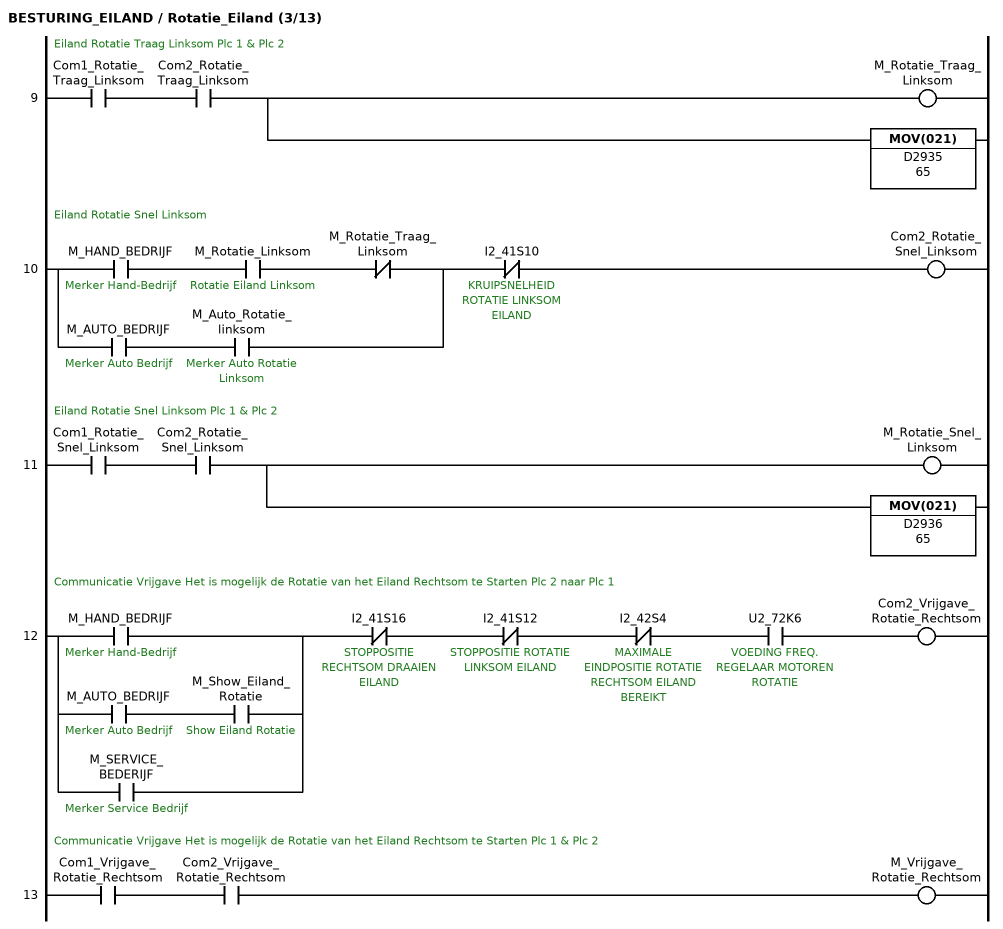
; [picture p421: BESTURING_EILAND / Rotatie_Eiland, rungs 9-13]
; rung 9: Eiland Rotatie Traag Linksom Plc 1 & Plc 2
LD Com1_Rotatie_Traag_Linksom
AND Com2_Rotatie_Traag_Linksom
OUT M_Rotatie_Traag_Linksom
MOV(021) D2935 65
; rung 10: Eiland Rotatie Snel Linksom
LD M_HAND_BEDRIJF  ; Merker Hand-Bedrijf
AND M_Rotatie_Linksom  ; Rotatie Eiland Linksom
ANDNOT M_Rotatie_Traag_Linksom
LD M_AUTO_BEDRIJF  ; Merker Auto Bedrijf
AND M_Auto_Rotatie_linksom  ; Merker Auto Rotatie Linksom
ORLD
ANDNOT I2_41S10  ; KRUIPSNELHEID ROTATIE LINKSOM EILAND
OUT Com2_Rotatie_Snel_Linksom
; rung 11: Eiland Rotatie Snel Linksom Plc 1 & Plc 2
LD Com1_Rotatie_Snel_Linksom
AND Com2_Rotatie_Snel_Linksom
OUT M_Rotatie_Snel_Linksom
MOV(021) D2936 65
; rung 12: Communicatie Vrijgave Het is mogelijk de Rotatie van het Eiland Rechtsom te Starten Plc 2 naar Plc 1
LD M_HAND_BEDRIJF  ; Merker Hand-Bedrijf
LD M_AUTO_BEDRIJF  ; Merker Auto Bedrijf
AND M_Show_Eiland_Rotatie  ; Show Eiland Rotatie
ORLD
OR M_SERVICE_BEDERIJF  ; Merker Service Bedrijf
ANDNOT I2_41S16  ; STOPPOSITIE RECHTSOM DRAAIEN EILAND
ANDNOT I2_41S12  ; STOPPOSITIE ROTATIE LINKSOM EILAND
ANDNOT I2_42S4  ; MAXIMALE EINDPOSITIE ROTATIE RECHTSOM EILAND BEREIKT
AND U2_72K6  ; VOEDING FREQ.REGELAAR MOTOREN ROTATIE
OUT Com2_Vrijgave_Rotatie_Rechtsom
; rung 13: Communicatie Vrijgave Het is mogelijk de Rotatie van het Eiland Rechtsom te Starten Plc 1 & Plc 2
LD Com1_Vrijgave_Rotatie_Rechtsom
AND Com2_Vrijgave_Rotatie_Rechtsom
OUT M_Vrijgave_Rotatie_Rechtsom

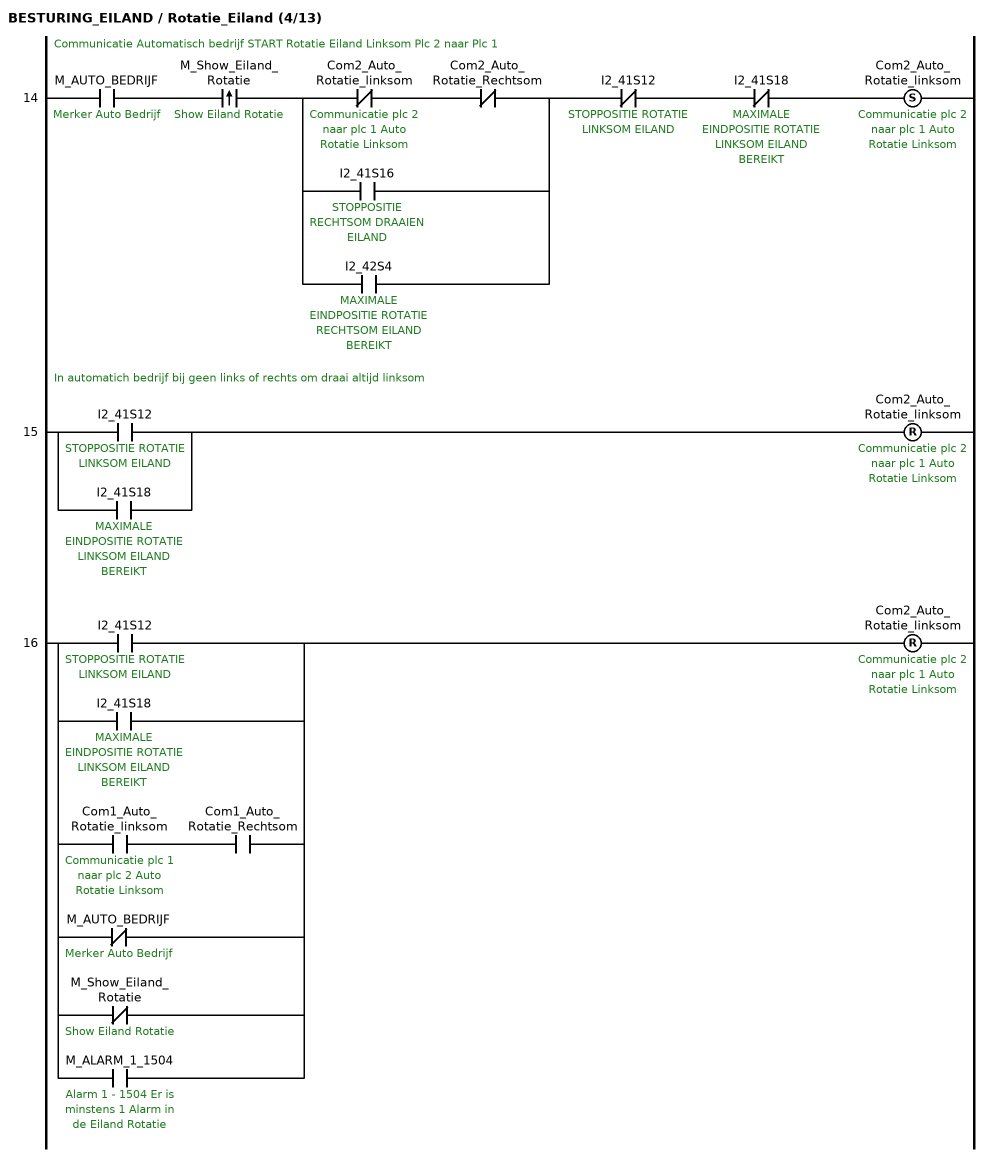
; rung 14: Communicatie Automatisch bedrijf START Rotatie Eiland Linksom Plc 2 naar Plc 1
LD M_AUTO_BEDRIJF  ; Merker Auto Bedrijf
@AND M_Show_Eiland_Rotatie  ; Show Eiland Rotatie
LDNOT Com2_Auto_Rotatie_linksom  ; Communicatie plc 2 naar plc 1 Auto Rotatie Linksom
ANDNOT Com2_Auto_Rotatie_Rechtsom
OR I2_41S16  ; STOPPOSITIE RECHTSOM DRAAIEN EILAND
OR I2_42S4  ; MAXIMALE EINDPOSITIE ROTATIE RECHTSOM EILAND BEREIKT
ANDLD
ANDNOT I2_41S12  ; STOPPOSITIE ROTATIE LINKSOM EILAND
ANDNOT I2_41S18  ; MAXIMALE EINDPOSITIE ROTATIE LINKSOM EILAND BEREIKT
SET Com2_Auto_Rotatie_linksom  ; Communicatie plc 2 naar plc 1 Auto Rotatie Linksom
; rung 15: In automatich bedrijf bij geen links of rechts om draai altijd linksom
LD I2_41S12  ; STOPPOSITIE ROTATIE LINKSOM EILAND
OR I2_41S18  ; MAXIMALE EINDPOSITIE ROTATIE LINKSOM EILAND BEREIKT
RSET Com2_Auto_Rotatie_linksom  ; Communicatie plc 2 naar plc 1 Auto Rotatie Linksom
; rung 16
LD I2_41S12  ; STOPPOSITIE ROTATIE LINKSOM EILAND
OR I2_41S18  ; MAXIMALE EINDPOSITIE ROTATIE LINKSOM EILAND BEREIKT
LD Com1_Auto_Rotatie_linksom  ; Communicatie plc 1 naar plc 2 Auto Rotatie Linksom
AND Com1_Auto_Rotatie_Rechtsom
ORLD
ORNOT M_AUTO_BEDRIJF  ; Merker Auto Bedrijf
ORNOT M_Show_Eiland_Rotatie  ; Show Eiland Rotatie
OR M_ALARM_1_1504  ; Alarm 1 - 1504 Er is minstens 1 Alarm in de Eiland Rotatie
RSET Com2_Auto_Rotatie_linksom  ; Communicatie plc 2 naar plc 1 Auto Rotatie Linksom

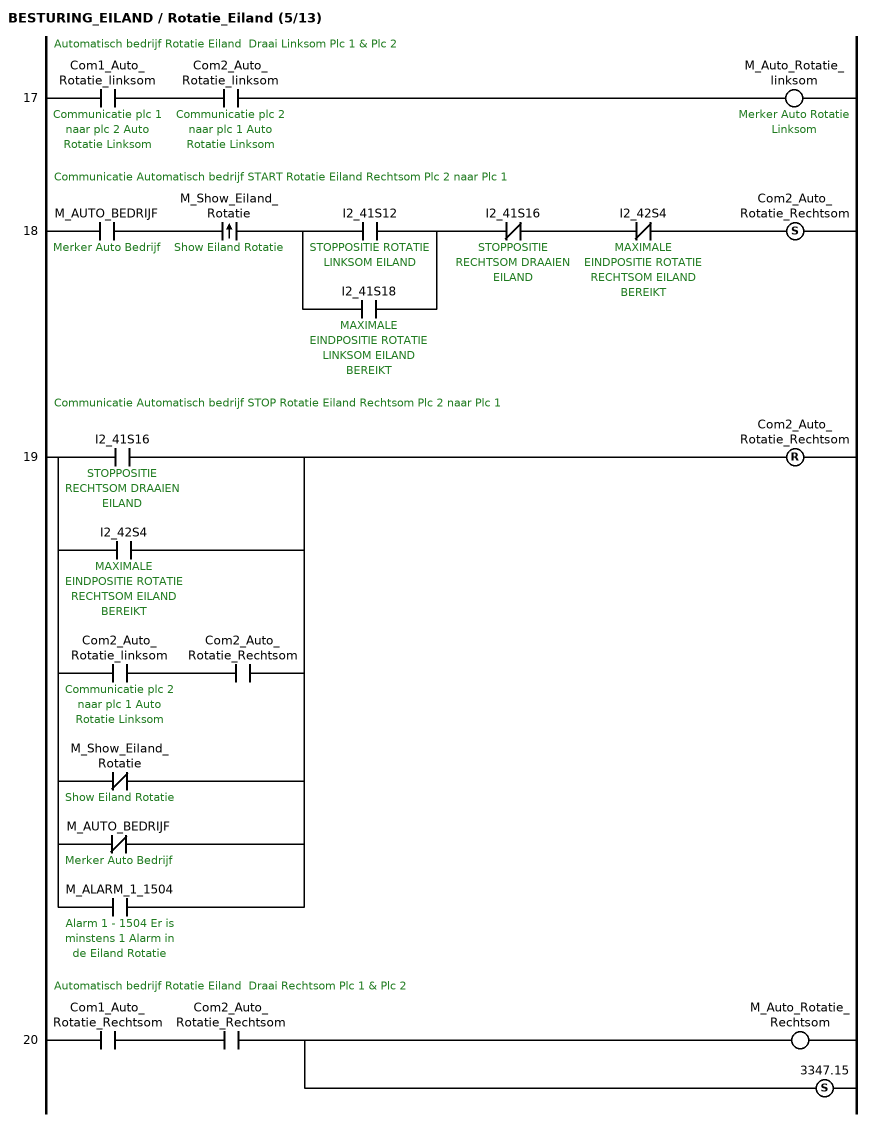
; rung 17: Automatisch bedrijf Rotatie Eiland  Draai Linksom Plc 1 & Plc 2
LD Com1_Auto_Rotatie_linksom  ; Communicatie plc 1 naar plc 2 Auto Rotatie Linksom
AND Com2_Auto_Rotatie_linksom  ; Communicatie plc 2 naar plc 1 Auto Rotatie Linksom
OUT M_Auto_Rotatie_linksom  ; Merker Auto Rotatie Linksom
; rung 18: Communicatie Automatisch bedrijf START Rotatie Eiland Rechtsom Plc 2 naar Plc 1
LD M_AUTO_BEDRIJF  ; Merker Auto Bedrijf
@AND M_Show_Eiland_Rotatie  ; Show Eiland Rotatie
LD I2_41S12  ; STOPPOSITIE ROTATIE LINKSOM EILAND
OR I2_41S18  ; MAXIMALE EINDPOSITIE ROTATIE LINKSOM EILAND BEREIKT
ANDLD
ANDNOT I2_41S16  ; STOPPOSITIE RECHTSOM DRAAIEN EILAND
ANDNOT I2_42S4  ; MAXIMALE EINDPOSITIE ROTATIE RECHTSOM EILAND BEREIKT
SET Com2_Auto_Rotatie_Rechtsom
; rung 19: Communicatie Automatisch bedrijf STOP Rotatie Eiland Rechtsom Plc 2 naar Plc 1
LD I2_41S16  ; STOPPOSITIE RECHTSOM DRAAIEN EILAND
OR I2_42S4  ; MAXIMALE EINDPOSITIE ROTATIE RECHTSOM EILAND BEREIKT
LD Com2_Auto_Rotatie_linksom  ; Communicatie plc 2 naar plc 1 Auto Rotatie Linksom
AND Com2_Auto_Rotatie_Rechtsom
ORLD
ORNOT M_Show_Eiland_Rotatie  ; Show Eiland Rotatie
ORNOT M_AUTO_BEDRIJF  ; Merker Auto Bedrijf
OR M_ALARM_1_1504  ; Alarm 1 - 1504 Er is minstens 1 Alarm in de Eiland Rotatie
RSET Com2_Auto_Rotatie_Rechtsom
; rung 20: Automatisch bedrijf Rotatie Eiland  Draai Rechtsom Plc 1 & Plc 2
LD Com1_Auto_Rotatie_Rechtsom
AND Com2_Auto_Rotatie_Rechtsom
OUT M_Auto_Rotatie_Rechtsom
SET 3347.15

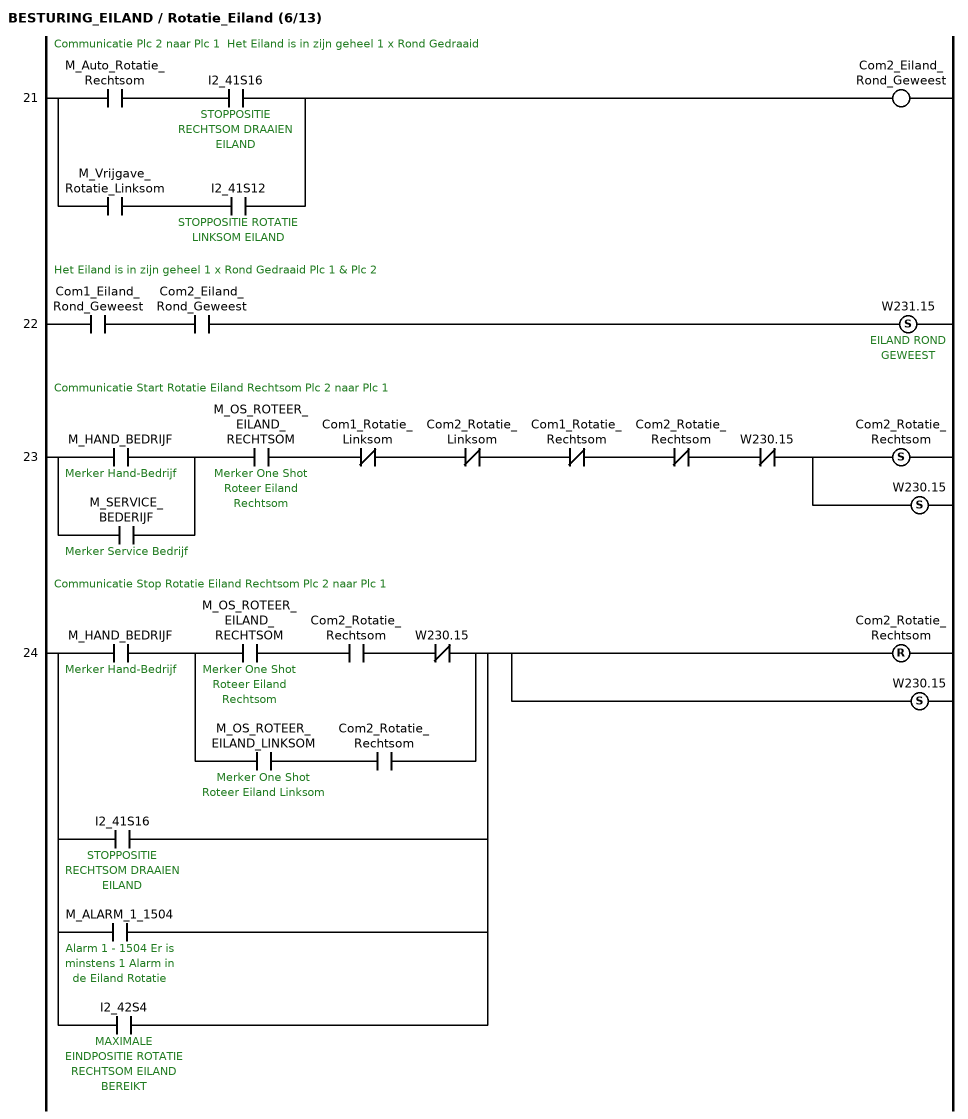
; rung 21: Communicatie Plc 2 naar Plc 1  Het Eiland is in zijn geheel 1 x Rond Gedraaid
LD M_Auto_Rotatie_Rechtsom
AND I2_41S16  ; STOPPOSITIE RECHTSOM DRAAIEN EILAND
LD M_Vrijgave_Rotatie_Linksom
AND I2_41S12  ; STOPPOSITIE ROTATIE LINKSOM EILAND
ORLD
OUT Com2_Eiland_Rond_Geweest
; rung 22: Het Eiland is in zijn geheel 1 x Rond Gedraaid Plc 1 & Plc 2
LD Com1_Eiland_Rond_Geweest
AND Com2_Eiland_Rond_Geweest
SET W231.15  ; EILAND ROND GEWEEST
; rung 23: Communicatie Start Rotatie Eiland Rechtsom Plc 2 naar Plc 1
LD M_HAND_BEDRIJF  ; Merker Hand-Bedrijf
OR M_SERVICE_BEDERIJF  ; Merker Service Bedrijf
AND M_OS_ROTEER_EILAND_RECHTSOM  ; Merker One Shot Roteer Eiland Rechtsom
ANDNOT Com1_Rotatie_Linksom
ANDNOT Com2_Rotatie_Linksom
ANDNOT Com1_Rotatie_Rechtsom
ANDNOT Com2_Rotatie_Rechtsom
ANDNOT W230.15
SET Com2_Rotatie_Rechtsom
SET W230.15
; rung 24: Communicatie Stop Rotatie Eiland Rechtsom Plc 2 naar Plc 1
LD M_HAND_BEDRIJF  ; Merker Hand-Bedrijf
LD M_OS_ROTEER_EILAND_RECHTSOM  ; Merker One Shot Roteer Eiland Rechtsom
AND Com2_Rotatie_Rechtsom
ANDNOT W230.15
LD M_OS_ROTEER_EILAND_LINKSOM  ; Merker One Shot Roteer Eiland Linksom
AND Com2_Rotatie_Rechtsom
ORLD
ANDLD
OR I2_41S16  ; STOPPOSITIE RECHTSOM DRAAIEN EILAND
OR M_ALARM_1_1504  ; Alarm 1 - 1504 Er is minstens 1 Alarm in de Eiland Rotatie
OR I2_42S4  ; MAXIMALE EINDPOSITIE ROTATIE RECHTSOM EILAND BEREIKT
RSET Com2_Rotatie_Rechtsom
SET W230.15

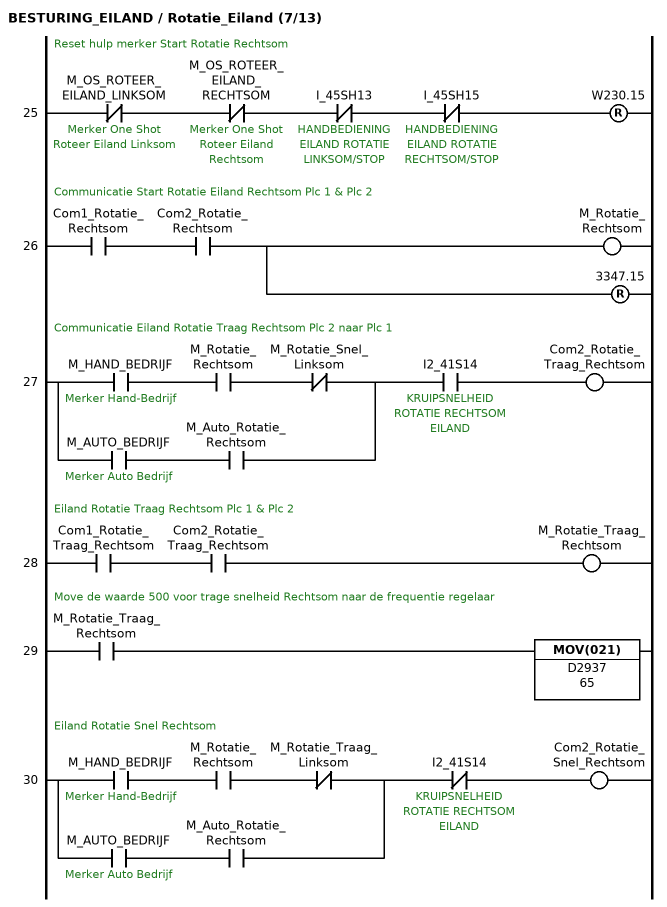
; rung 25: Reset hulp merker Start Rotatie Rechtsom
LDNOT M_OS_ROTEER_EILAND_LINKSOM  ; Merker One Shot Roteer Eiland Linksom
ANDNOT M_OS_ROTEER_EILAND_RECHTSOM  ; Merker One Shot Roteer Eiland Rechtsom
ANDNOT I_45SH13  ; HANDBEDIENING EILAND ROTATIE LINKSOM/STOP
ANDNOT I_45SH15  ; HANDBEDIENING EILAND ROTATIE RECHTSOM/STOP
RSET W230.15
; rung 26: Communicatie Start Rotatie Eiland Rechtsom Plc 1 & Plc 2
LD Com1_Rotatie_Rechtsom
AND Com2_Rotatie_Rechtsom
OUT M_Rotatie_Rechtsom
RSET 3347.15
; rung 27: Communicatie Eiland Rotatie Traag Rechtsom Plc 2 naar Plc 1
LD M_HAND_BEDRIJF  ; Merker Hand-Bedrijf
AND M_Rotatie_Rechtsom
ANDNOT M_Rotatie_Snel_Linksom
LD M_AUTO_BEDRIJF  ; Merker Auto Bedrijf
AND M_Auto_Rotatie_Rechtsom
ORLD
AND I2_41S14  ; KRUIPSNELHEID ROTATIE RECHTSOM EILAND
OUT Com2_Rotatie_Traag_Rechtsom
; rung 28: Eiland Rotatie Traag Rechtsom Plc 1 & Plc 2
LD Com1_Rotatie_Traag_Rechtsom
AND Com2_Rotatie_Traag_Rechtsom
OUT M_Rotatie_Traag_Rechtsom
; rung 29: Move de waarde 500 voor trage snelheid Rechtsom naar de frequentie regelaar
LD M_Rotatie_Traag_Rechtsom
MOV(021) D2937 65
; rung 30: Eiland Rotatie Snel Rechtsom
LD M_HAND_BEDRIJF  ; Merker Hand-Bedrijf
AND M_Rotatie_Rechtsom
ANDNOT M_Rotatie_Traag_Linksom
LD M_AUTO_BEDRIJF  ; Merker Auto Bedrijf
AND M_Auto_Rotatie_Rechtsom
ORLD
ANDNOT I2_41S14  ; KRUIPSNELHEID ROTATIE RECHTSOM EILAND
OUT Com2_Rotatie_Snel_Rechtsom

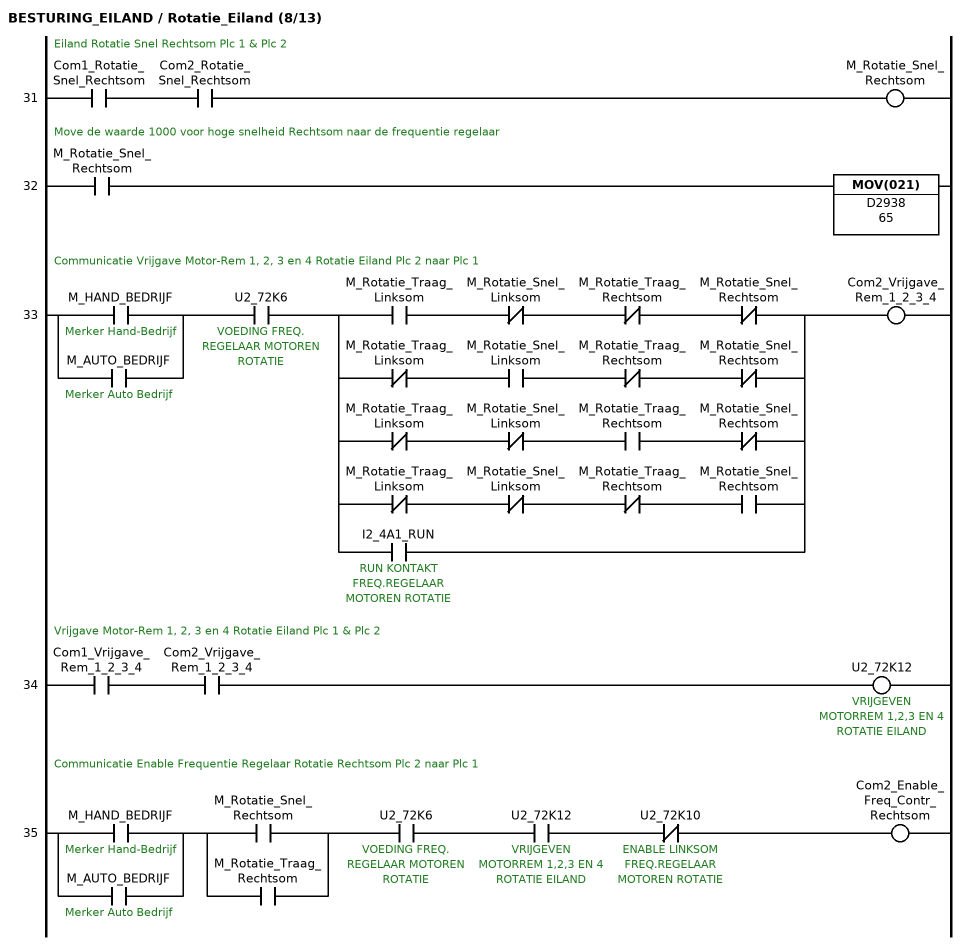
; rung 31: Eiland Rotatie Snel Rechtsom Plc 1 & Plc 2
LD Com1_Rotatie_Snel_Rechtsom
AND Com2_Rotatie_Snel_Rechtsom
OUT M_Rotatie_Snel_Rechtsom
; rung 32: Move de waarde 1000 voor hoge snelheid Rechtsom naar de frequentie regelaar
LD M_Rotatie_Snel_Rechtsom
MOV(021) D2938 65
; rung 33: Communicatie Vrijgave Motor-Rem 1, 2, 3 en 4 Rotatie Eiland Plc 2 naar Plc 1
LD M_HAND_BEDRIJF  ; Merker Hand-Bedrijf
OR M_AUTO_BEDRIJF  ; Merker Auto Bedrijf
AND U2_72K6  ; VOEDING FREQ.REGELAAR MOTOREN ROTATIE
LD M_Rotatie_Traag_Linksom
ANDNOT M_Rotatie_Snel_Linksom
ANDNOT M_Rotatie_Traag_Rechtsom
ANDNOT M_Rotatie_Snel_Rechtsom
LDNOT M_Rotatie_Traag_Linksom
AND M_Rotatie_Snel_Linksom
ANDNOT M_Rotatie_Traag_Rechtsom
ANDNOT M_Rotatie_Snel_Rechtsom
ORLD
LDNOT M_Rotatie_Traag_Linksom
ANDNOT M_Rotatie_Snel_Linksom
AND M_Rotatie_Traag_Rechtsom
ANDNOT M_Rotatie_Snel_Rechtsom
ORLD
LDNOT M_Rotatie_Traag_Linksom
ANDNOT M_Rotatie_Snel_Linksom
ANDNOT M_Rotatie_Traag_Rechtsom
AND M_Rotatie_Snel_Rechtsom
ORLD
OR I2_4A1_RUN  ; RUN KONTAKT FREQ.REGELAAR MOTOREN ROTATIE
ANDLD
OUT Com2_Vrijgave_Rem_1_2_3_4
; rung 34: Vrijgave Motor-Rem 1, 2, 3 en 4 Rotatie Eiland Plc 1 & Plc 2
LD Com1_Vrijgave_Rem_1_2_3_4
AND Com2_Vrijgave_Rem_1_2_3_4
OUT U2_72K12  ; VRIJGEVEN MOTORREM 1,2,3 EN 4 ROTATIE EILAND
; rung 35: Communicatie Enable Frequentie Regelaar Rotatie Rechtsom Plc 2 naar Plc 1
LD M_HAND_BEDRIJF  ; Merker Hand-Bedrijf
OR M_AUTO_BEDRIJF  ; Merker Auto Bedrijf
LD M_Rotatie_Snel_Rechtsom
OR M_Rotatie_Traag_Rechtsom
ANDLD
AND U2_72K6  ; VOEDING FREQ.REGELAAR MOTOREN ROTATIE
AND U2_72K12  ; VRIJGEVEN MOTORREM 1,2,3 EN 4 ROTATIE EILAND
ANDNOT U2_72K10  ; ENABLE LINKSOM FREQ.REGELAAR MOTOREN ROTATIE
OUT Com2_Enable_Freq_Contr_Rechtsom

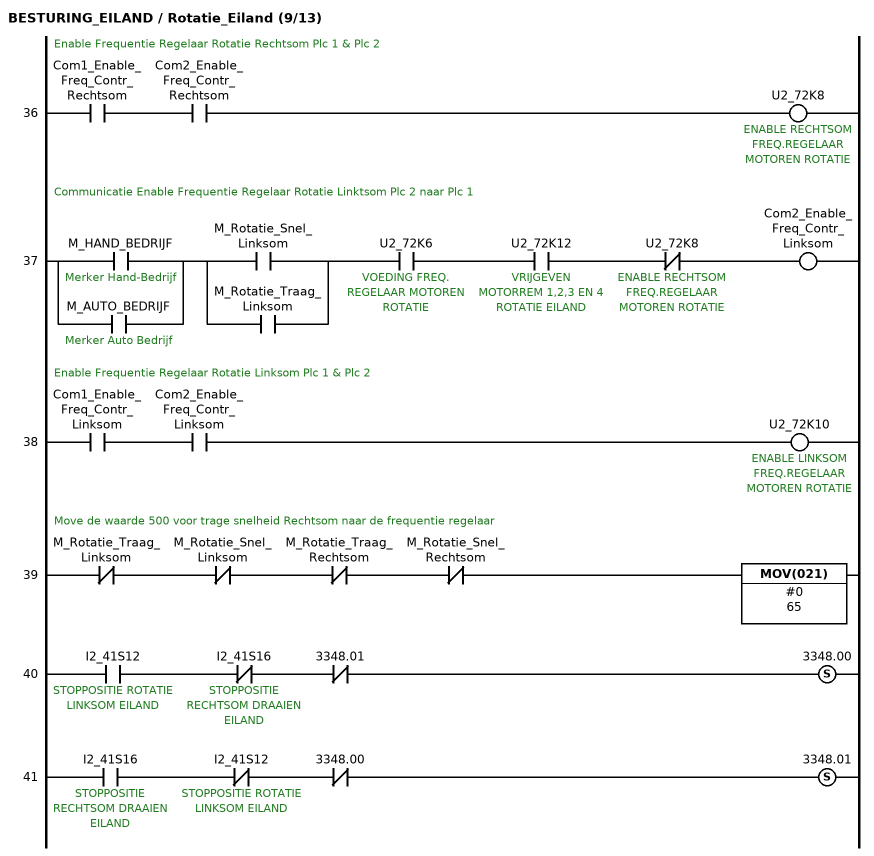
; rung 36: Enable Frequentie Regelaar Rotatie Rechtsom Plc 1 & Plc 2
LD Com1_Enable_Freq_Contr_Rechtsom
AND Com2_Enable_Freq_Contr_Rechtsom
OUT U2_72K8  ; ENABLE RECHTSOM FREQ.REGELAAR MOTOREN ROTATIE
; rung 37: Communicatie Enable Frequentie Regelaar Rotatie Linktsom Plc 2 naar Plc 1
LD M_HAND_BEDRIJF  ; Merker Hand-Bedrijf
OR M_AUTO_BEDRIJF  ; Merker Auto Bedrijf
LD M_Rotatie_Snel_Linksom
OR M_Rotatie_Traag_Linksom
ANDLD
AND U2_72K6  ; VOEDING FREQ.REGELAAR MOTOREN ROTATIE
AND U2_72K12  ; VRIJGEVEN MOTORREM 1,2,3 EN 4 ROTATIE EILAND
ANDNOT U2_72K8  ; ENABLE RECHTSOM FREQ.REGELAAR MOTOREN ROTATIE
OUT Com2_Enable_Freq_Contr_Linksom
; rung 38: Enable Frequentie Regelaar Rotatie Linksom Plc 1 & Plc 2
LD Com1_Enable_Freq_Contr_Linksom
AND Com2_Enable_Freq_Contr_Linksom
OUT U2_72K10  ; ENABLE LINKSOM FREQ.REGELAAR MOTOREN ROTATIE
; rung 39: Move de waarde 500 voor trage snelheid Rechtsom naar de frequentie regelaar
LDNOT M_Rotatie_Traag_Linksom
ANDNOT M_Rotatie_Snel_Linksom
ANDNOT M_Rotatie_Traag_Rechtsom
ANDNOT M_Rotatie_Snel_Rechtsom
MOV(021) #0 65
; rung 40
LD I2_41S12  ; STOPPOSITIE ROTATIE LINKSOM EILAND
ANDNOT I2_41S16  ; STOPPOSITIE RECHTSOM DRAAIEN EILAND
ANDNOT 3348.01
SET 3348.00
; rung 41
LD I2_41S16  ; STOPPOSITIE RECHTSOM DRAAIEN EILAND
ANDNOT I2_41S12  ; STOPPOSITIE ROTATIE LINKSOM EILAND
ANDNOT 3348.00
SET 3348.01

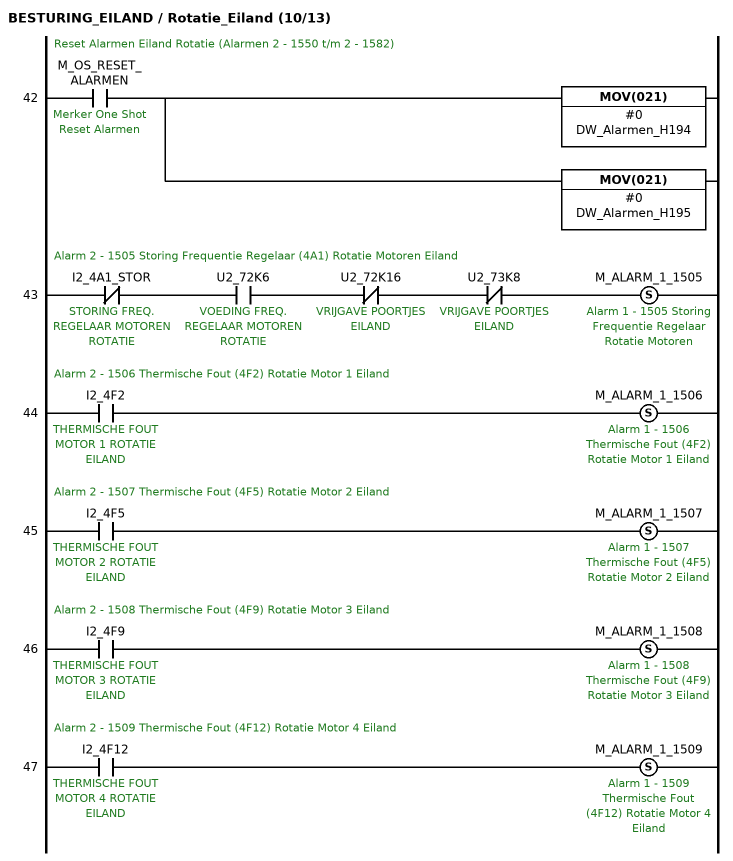
; rung 42: Reset Alarmen Eiland Rotatie (Alarmen 2 - 1550 t/m 2 - 1582)
LD M_OS_RESET_ALARMEN  ; Merker One Shot Reset Alarmen
MOV(021) #0 DW_Alarmen_H194
MOV(021) #0 DW_Alarmen_H195
; rung 43: Alarm 2 - 1505 Storing Frequentie Regelaar (4A1) Rotatie Motoren Eiland
LDNOT I2_4A1_STOR  ; STORING FREQ.REGELAAR MOTOREN ROTATIE
AND U2_72K6  ; VOEDING FREQ.REGELAAR MOTOREN ROTATIE
ANDNOT U2_72K16  ; VRIJGAVE POORTJES EILAND
ANDNOT U2_73K8  ; VRIJGAVE POORTJES EILAND
SET M_ALARM_1_1505  ; Alarm 1 - 1505 Storing Frequentie Regelaar Rotatie Motoren
; rung 44: Alarm 2 - 1506 Thermische Fout (4F2) Rotatie Motor 1 Eiland
LD I2_4F2  ; THERMISCHE FOUT MOTOR 1 ROTATIE EILAND
SET M_ALARM_1_1506  ; Alarm 1 - 1506 Thermische Fout (4F2) Rotatie Motor 1 Eiland
; rung 45: Alarm 2 - 1507 Thermische Fout (4F5) Rotatie Motor 2 Eiland
LD I2_4F5  ; THERMISCHE FOUT MOTOR 2 ROTATIE EILAND
SET M_ALARM_1_1507  ; Alarm 1 - 1507 Thermische Fout (4F5) Rotatie Motor 2 Eiland
; rung 46: Alarm 2 - 1508 Thermische Fout (4F9) Rotatie Motor 3 Eiland
LD I2_4F9  ; THERMISCHE FOUT MOTOR 3 ROTATIE EILAND
SET M_ALARM_1_1508  ; Alarm 1 - 1508 Thermische Fout (4F9) Rotatie Motor 3 Eiland
; rung 47: Alarm 2 - 1509 Thermische Fout (4F12) Rotatie Motor 4 Eiland
LD I2_4F12  ; THERMISCHE FOUT MOTOR 4 ROTATIE EILAND
SET M_ALARM_1_1509  ; Alarm 1 - 1509 Thermische Fout (4F12) Rotatie Motor 4 Eiland

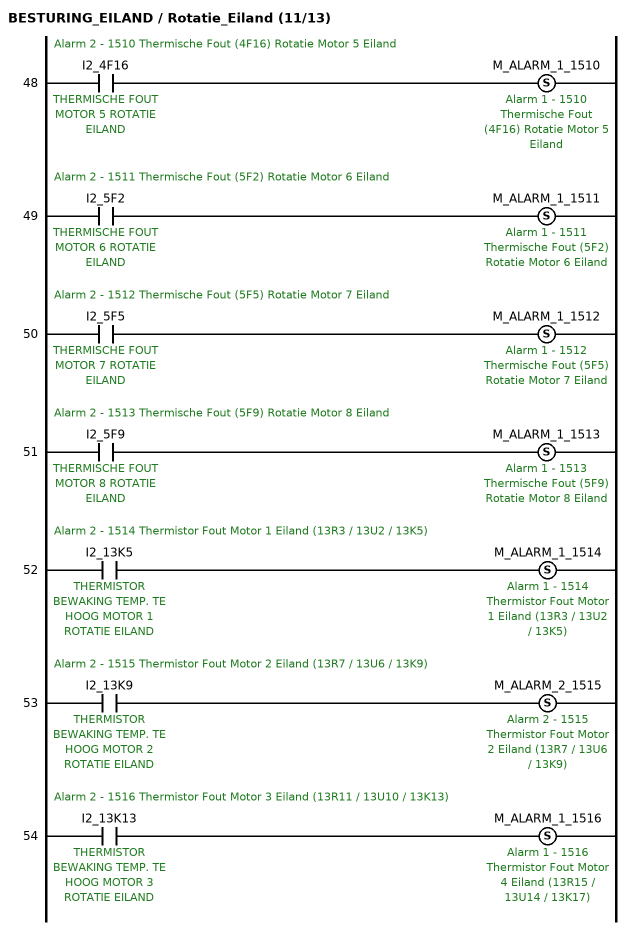
; rung 48: Alarm 2 - 1510 Thermische Fout (4F16) Rotatie Motor 5 Eiland
LD I2_4F16  ; THERMISCHE FOUT MOTOR 5 ROTATIE EILAND
SET M_ALARM_1_1510  ; Alarm 1 - 1510 Thermische Fout (4F16) Rotatie Motor 5 Eiland
; rung 49: Alarm 2 - 1511 Thermische Fout (5F2) Rotatie Motor 6 Eiland
LD I2_5F2  ; THERMISCHE FOUT MOTOR 6 ROTATIE EILAND
SET M_ALARM_1_1511  ; Alarm 1 - 1511 Thermische Fout (5F2) Rotatie Motor 6 Eiland
; rung 50: Alarm 2 - 1512 Thermische Fout (5F5) Rotatie Motor 7 Eiland
LD I2_5F5  ; THERMISCHE FOUT MOTOR 7 ROTATIE EILAND
SET M_ALARM_1_1512  ; Alarm 1 - 1512 Thermische Fout (5F5) Rotatie Motor 7 Eiland
; rung 51: Alarm 2 - 1513 Thermische Fout (5F9) Rotatie Motor 8 Eiland
LD I2_5F9  ; THERMISCHE FOUT MOTOR 8 ROTATIE EILAND
SET M_ALARM_1_1513  ; Alarm 1 - 1513 Thermische Fout (5F9) Rotatie Motor 8 Eiland
; rung 52: Alarm 2 - 1514 Thermistor Fout Motor 1 Eiland (13R3 / 13U2 / 13K5)
LD I2_13K5  ; THERMISTOR BEWAKING TEMP. TE HOOG MOTOR 1 ROTATIE EILAND
SET M_ALARM_1_1514  ; Alarm 1 - 1514 Thermistor Fout Motor 1 Eiland (13R3 / 13U2 / 13K5)
; rung 53: Alarm 2 - 1515 Thermistor Fout Motor 2 Eiland (13R7 / 13U6 / 13K9)
LD I2_13K9  ; THERMISTOR BEWAKING TEMP. TE HOOG MOTOR 2 ROTATIE EILAND
SET M_ALARM_2_1515  ; Alarm 2 - 1515 Thermistor Fout Motor 2 Eiland (13R7 / 13U6 / 13K9)
; rung 54: Alarm 2 - 1516 Thermistor Fout Motor 3 Eiland (13R11 / 13U10 / 13K13)
LD I2_13K13  ; THERMISTOR BEWAKING TEMP. TE HOOG MOTOR 3 ROTATIE EILAND
SET M_ALARM_1_1516  ; Alarm 1 - 1516 Thermistor Fout Motor 4 Eiland (13R15 / 13U14 / 13K17)

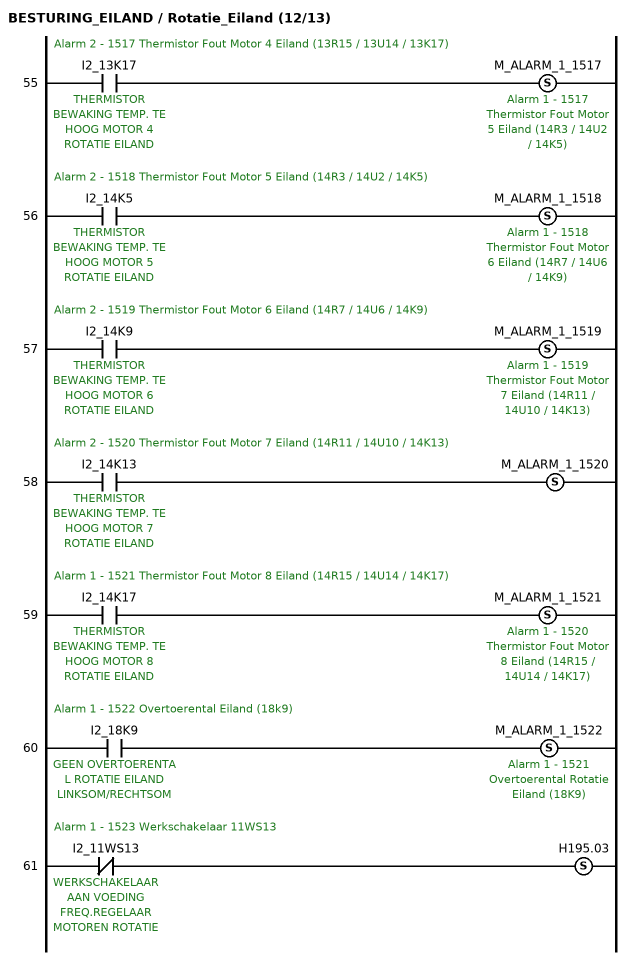
; rung 55: Alarm 2 - 1517 Thermistor Fout Motor 4 Eiland (13R15 / 13U14 / 13K17)
LD I2_13K17  ; THERMISTOR BEWAKING TEMP. TE HOOG MOTOR 4 ROTATIE EILAND
SET M_ALARM_1_1517  ; Alarm 1 - 1517 Thermistor Fout Motor 5 Eiland (14R3 / 14U2 / 14K5)
; rung 56: Alarm 2 - 1518 Thermistor Fout Motor 5 Eiland (14R3 / 14U2 / 14K5)
LD I2_14K5  ; THERMISTOR BEWAKING TEMP. TE HOOG MOTOR 5 ROTATIE EILAND
SET M_ALARM_1_1518  ; Alarm 1 - 1518 Thermistor Fout Motor 6 Eiland (14R7 / 14U6 / 14K9)
; rung 57: Alarm 2 - 1519 Thermistor Fout Motor 6 Eiland (14R7 / 14U6 / 14K9)
LD I2_14K9  ; THERMISTOR BEWAKING TEMP. TE HOOG MOTOR 6 ROTATIE EILAND
SET M_ALARM_1_1519  ; Alarm 1 - 1519 Thermistor Fout Motor 7 Eiland (14R11 / 14U10 / 14K13)
; rung 58: Alarm 2 - 1520 Thermistor Fout Motor 7 Eiland (14R11 / 14U10 / 14K13)
LD I2_14K13  ; THERMISTOR BEWAKING TEMP. TE HOOG MOTOR 7 ROTATIE EILAND
SET M_ALARM_1_1520
; rung 59: Alarm 1 - 1521 Thermistor Fout Motor 8 Eiland (14R15 / 14U14 / 14K17)
LD I2_14K17  ; THERMISTOR BEWAKING TEMP. TE HOOG MOTOR 8 ROTATIE EILAND
SET M_ALARM_1_1521  ; Alarm 1 - 1520 Thermistor Fout Motor 8 Eiland (14R15 / 14U14 / 14K17)
; rung 60: Alarm 1 - 1522 Overtoerental Eiland (18k9)
LD I2_18K9  ; GEEN OVERTOERENTAL ROTATIE EILAND LINKSOM/RECHTSOM
SET M_ALARM_1_1522  ; Alarm 1 - 1521 Overtoerental Rotatie Eiland (18K9)
; rung 61: Alarm 1 - 1523 Werkschakelaar 11WS13
LDNOT I2_11WS13  ; WERKSCHAKELAAR AAN VOEDING FREQ.REGELAAR MOTOREN ROTATIE
SET H195.03

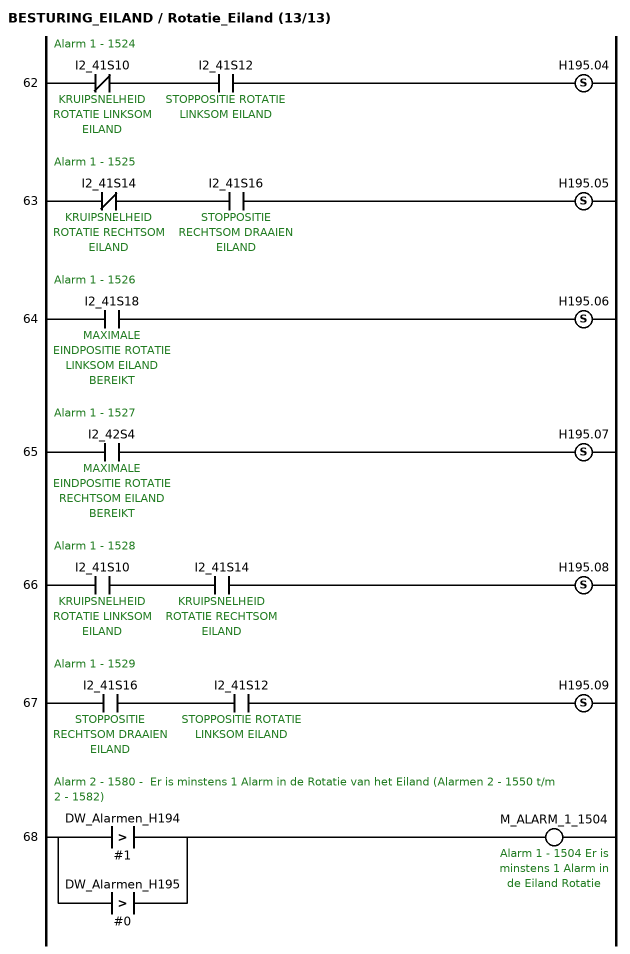
; rung 62: Alarm 1 - 1524
LDNOT I2_41S10  ; KRUIPSNELHEID ROTATIE LINKSOM EILAND
AND I2_41S12  ; STOPPOSITIE ROTATIE LINKSOM EILAND
SET H195.04
; rung 63: Alarm 1 - 1525
LDNOT I2_41S14  ; KRUIPSNELHEID ROTATIE RECHTSOM EILAND
AND I2_41S16  ; STOPPOSITIE RECHTSOM DRAAIEN EILAND
SET H195.05
; rung 64: Alarm 1 - 1526
LD I2_41S18  ; MAXIMALE EINDPOSITIE ROTATIE LINKSOM EILAND BEREIKT
SET H195.06
; rung 65: Alarm 1 - 1527
LD I2_42S4  ; MAXIMALE EINDPOSITIE ROTATIE RECHTSOM EILAND BEREIKT
SET H195.07
; rung 66: Alarm 1 - 1528
LD I2_41S10  ; KRUIPSNELHEID ROTATIE LINKSOM EILAND
AND I2_41S14  ; KRUIPSNELHEID ROTATIE RECHTSOM EILAND
SET H195.08
; rung 67: Alarm 1 - 1529
LD I2_41S16  ; STOPPOSITIE RECHTSOM DRAAIEN EILAND
AND I2_41S12  ; STOPPOSITIE ROTATIE LINKSOM EILAND
SET H195.09
; rung 68: Alarm 2 - 1580 -  Er is minstens 1 Alarm in de Rotatie van het Eiland (Alarmen 2 - 1550 t/m 2 - 1582)
LD>(320) DW_Alarmen_H194 #1
OR>(320) DW_Alarmen_H195 #0
OUT M_ALARM_1_1504  ; Alarm 1 - 1504 Er is minstens 1 Alarm in de Eiland Rotatie

### Section EInde_Besturing_Eiland
; rung 0
END(001)

# PLC PLC3_PAGODE_EILAND: CJ2M CPU12
I/O table (CPU CJ2M-CPU12): rack 0 slot 0 CJ1W-CLK23; rack 0 slot 1 CJ1W-ID211; rack 0 slot 2 CJ1W-ID211; rack 0 slot 3 CJ1W-ID211; rack 0 slot 4 CJ1W-ID211; rack 0 slot 5 CJ1W-OD212; rack 0 slot 6 CJ1W-OD212; rack 0 slot 7 CJ1W-OD212

## Global symbols (name address type ; comment)
ALL_24_VDC_RELAY_ON 230.03 BOOL  ; ALL 24 VDC RELAY ON
102.01 BOOL  ; show afbreken
102.02 BOOL  ; noodberging 1
102.03 BOOL  ; noodberging 2
125.03 BOOL  ; Signalering stop show vanaf grond
217.00 BOOL  ; Alarm in register 0 zoeken
217.01 BOOL  ; Alarm in register 1 zoeken
217.02 BOOL  ; Alarm in register 2 zoeken
217.03 BOOL  ; Alarm in register 3 zoeken
217.04 BOOL  ; Alarm in register 4 zoeken
217.05 BOOL  ; Alarm in register 5 zoeken
217.08 BOOL  ; Alarm (1 of meerdere)
217.09 BOOL  ; Alarmlamp knipperen bij nieuw alarm
217.10 BOOL  ; Zoeken naar nieuw alarm
217.11 BOOL  ; Volgend alarmwoord bekijken
217.12 BOOL  ; Alarm zoeken in volgende woord
217.13 BOOL  ; Volgende alarm gevonden
217.14 BOOL  ; Elke 2 seconden 1 scan hoog
217.15 BOOL  ; Zoek volgende alarm melding
218.08 BOOL  ; Nieuw alarm in woord HR30
218.09 BOOL  ; Nieuw alarm in woord HR31
218.10 BOOL  ; Nieuw alarm in woord HR32
218.11 BOOL  ; Nieuw alarm in woord HR33
218.12 BOOL  ; Nieuw alarm in woord HR34
218.13 BOOL  ; Nieuw alarm in woord HR35
218.14 BOOL  ; Geen nieuw alarm
218.15 BOOL  ; 1 scan, er is een nieuw alarm opgetreden
219.00 BOOL  ; Alarm in register 6 zoeken
219.01 BOOL  ; Alarm in register 7 zoeken
219.02 BOOL  ; Alarm in register 8 zoeken
219.03 BOOL  ; Alarm in register 8 zoeken
219.08 BOOL  ; Nieuw alarm in woord HR36
219.09 BOOL  ; Nieuw alarm in woord HR37
219.10 BOOL  ; Nieuw alarm in woord HR38
219.11 BOOL  ; Alle poorten staan dicht
224.00 BOOL  ; Poort 1 links is open
224.01 BOOL  ; Poort 1 links is dicht
224.02 BOOL  ; Poort 1 links is aan het openen
224.03 BOOL  ; Poort 1 links is aan het sluiten
224.04 BOOL  ; Poort 1 rechts is open
224.05 BOOL  ; Poort 1 rechts is dicht
224.06 BOOL  ; Poort 1 rechts is aan het openen
224.07 BOOL  ; Poort 1 rechts is aan het sluiten
224.08 BOOL  ; Poort 2 links is open
224.09 BOOL  ; Poort 2 links is dicht
224.10 BOOL  ; Poort 2 links is aan het openen
224.11 BOOL  ; poort 2 links is aan het sluiten
224.12 BOOL  ; Poort 2 rechts is open
224.13 BOOL  ; Poort 2 rechts is dicht
224.14 BOOL  ; Poort 2 rechts is aan het openen
224.15 BOOL  ; Poort 2 rechts is aan het sluiten
225.00 BOOL  ; Poort 3 links is open
225.01 BOOL  ; Poort 3 links is dicht
225.02 BOOL  ; Poort 3 links is aan het openen
225.03 BOOL  ; Poort 3 links is aan het sluiten
225.04 BOOL  ; Poort 3 rechts is open
225.05 BOOL  ; Poort 3 rechts is dicht
225.06 BOOL  ; Poort 3 rechts is aan het openen
225.07 BOOL  ; Poort 3 rechts is aan het sluiten
225.08 BOOL  ; Poort 4 links is open
225.09 BOOL  ; Poort 4 links is dicht
225.10 BOOL  ; Poort 4 links is aan het openen
225.11 BOOL  ; Poort 4 links is aan het sluiten
225.12 BOOL  ; Poort 4 rechts is open
225.13 BOOL  ; Poort 4 rechts is dicht
225.14 BOOL  ; Poort 4 rechts is aan het openen
225.15 BOOL  ; Poort 4 rechts is aan het sluiten
230.04 BOOL  ; stop show
232.02 BOOL  ; stop van grond
240.01 BOOL  ; Testmerker
T0100 BOOL  ; DISPATCH TIMER
T0101 BOOL  ; TIMER 24 VDC RELAY 01 (ALL RELAY ON)
T0102 BOOL  ; TIMER 24 VDC RELAY 02 (ONE RELAY OFF)
DISPATCH_ACTIVE 231.00 BOOL  ; DISPATCH ACTIVE
DISPATCH_ISLAND_ENABLE 230.00 BOOL  ; DISPATCH ISLAND ENABLE
DISPATCH_TIMER 100 NUMBER  ; DISPATCH TIMER
DISPATCH_TIMER_ACTIVE 230.02 BOOL  ; DISPATCH TIMER ACTIVE
I1L_BEWAK 2.08 BOOL  ; POORT 1 LINKS BEWAKING
I1L_BIJNA 0.07 BOOL  ; POORT 1 LINKS BIJNA DICHT
I1L_DICHT 0.06 BOOL  ; POORT 1 LINKS DICHT
I1L_GREND 2.00 BOOL  ; POORT 1 LINKS VERGRENDELD
I1L_OPEN 0.08 BOOL  ; POORT 1 LINKS OPEN
I1R_BEWAK 2.09 BOOL  ; POORT 1 RECHTS BEWAKING
I1R_BIJNA 0.10 BOOL  ; POORT 1 RECHTS BIJNA DICHT
I1R_DICHT 0.09 BOOL  ; POORT 1 RECHTS DICHT
I1R_GREND 2.01 BOOL  ; POORT 1 RECHTS VERGRENDELD
I1R_OPEN 0.11 BOOL  ; POORT 1 RECHTS OPEN
I24V_OKE1 3.00 BOOL  ; 24 VOLT OKE (MELDING 1)
I24V_OKE2 3.01 BOOL  ; 24 VOLT OKE (MELDING 2)
I24V_OKE3 3.02 BOOL  ; 24 VOLT OKE (MELDING 3)
I2L_BEWAK 2.10 BOOL  ; POORT 2 LINKS BEWAKING
I2L_BIJNA 0.13 BOOL  ; POORT 2 LINKS BIJNA DICHT
I2L_DICHT 0.12 BOOL  ; POORT 2 LINKS DICHT
I2L_GREND 2.02 BOOL  ; POORT 2 LINKS VERGRENDELD
I2L_OPEN 0.14 BOOL  ; POORT 2 LINKS OPEN
I2R_BEWAK 2.11 BOOL  ; POORT 2 RECHTS BEWAKING
I2R_BIJNA 1.00 BOOL  ; POORT 2 RECHTS BIJNA DICHT
I2R_DICHT 0.15 BOOL  ; POORT 2 RECHTS DICHT
I2R_GREND 2.03 BOOL  ; POORT 2 RECHTS VERGRENDELD
I2R_OPEN 1.01 BOOL  ; POORT 2 RECHTS OPEN
I3L_BEWAK 2.12 BOOL  ; POORT 3 LINKS BEWAKING
I3L_BIJNA 1.03 BOOL  ; POORT 3 LINKS  BIJNA DICHT
I3L_DICHT 1.02 BOOL  ; POORT 3 LINKS  DICHT
I3L_GREND 2.04 BOOL  ; POORT 3 LINKS VERGRENDELD
I3L_OPEN 1.04 BOOL  ; POORT 3 LINKS  OPEN
I3R_BEWAK 2.13 BOOL  ; POORT 3 RECHTS BEWAKING
I3R_BIJNA 1.06 BOOL  ; POORT 3 RECHTS BIJNA DICHT
I3R_DICHT 1.05 BOOL  ; POORT 3 RECHTS DICHT
I3R_GREND 2.05 BOOL  ; POORT 3 RECHTS VERGRENDELD
I3R_OPEN 1.07 BOOL  ; POORT 3 RECHTS OPEN
I4L_BEWAK 2.14 BOOL  ; POORT 4 LINKS BEWAKING
I4L_BIJNA 1.09 BOOL  ; POORT 4 LINKS BIJNA DICHT
I4L_DICHT 1.08 BOOL  ; POORT 4 LINKS DICHT
I4L_GREND 2.06 BOOL  ; POORT 4 LINKS VERGRENDELD
I4L_OPEN 1.10 BOOL  ; POORT 4 LINKS OPEN
I4R_BEWAK 2.15 BOOL  ; POORT 4 RECHTS BEWAKING
I4R_BIJNA 1.12 BOOL  ; POORT 4 RECHTS BIJNA DICHT
I4R_DICHT 1.11 BOOL  ; POORT 4 RECHTS DICHT
I4R_GREND 2.07 BOOL  ; POORT 4 RECHTS VERGRENDELD
I4R_OPEN 1.13 BOOL  ; POORT 4 RECHTS OPEN
IAUTOMAAT 0.05 BOOL  ; AUTOMAAT VOEDINGS GROEP MOTOREN
INIT_BIT A200.15 BOOL  ; FIRST SCAN BIT
INOODSTOP 0.00 BOOL  ; NOODSTOP OKE
IOPEN_IN 0.01 BOOL  ; DK OPENEN POORTEN INGANG
IOPEN_UI 0.03 BOOL  ; DK OPENEN POORTEN UITGANG
IREADY 1.14 BOOL  ; DK READY SIGNAAL
IRESET 1.15 BOOL  ; DK RESET
ISLUIT_IN 0.02 BOOL  ; DK SLUITEN POORTEN INGANG
ISLUIT_UI 0.04 BOOL  ; DK SLUITEN POORTEN UITGANG
M1SECPULS CF102 BOOL  ; 1 SEC. HOOG, 1 SEC LAAG = 0,5 HZ
MAL19909 27.09 BOOL  ; OUTPUT ALARM RESERVE BIT
MAL19910 27.10 BOOL  ; OUTPUT ALARM RESERVE BIT
MAL19911 27.11 BOOL  ; OUTPUT ALARM RESERVE BIT
MAL19912 27.12 BOOL  ; OUTPUT ALARM RESERVE BIT
MAL19913 27.13 BOOL  ; OUTPUT ALARM RESEREV BIT
MAL19914 27.14 BOOL  ; OUTPUT ALARM RESEREV BIT
MAL19915 27.15 BOOL  ; OUTPUT ALARM RESERVE BIT
MALBEWAK 27.08 BOOL  ; ALARM BEWAKING AANGESPROKEN
MALM9909 23.09 BOOL  ; ALARM RESERVE BIT
MALM9910 23.10 BOOL  ; ALARM RESERVE BIT
MALM9911 23.11 BOOL  ; ALARM RESERVE BIT
MALM9912 23.12 BOOL  ; ALARM RESERVE BIT
MALM9913 23.13 BOOL  ; ALARM RESERVE BIT
MALM9914 23.14 BOOL  ; ALARM RESERVE BIT
MALM9915 23.15 BOOL  ; ALARM RESERVE BIT
MALMBIJ1 27.04 BOOL  ; ALARM BIJNA OPEN SENSOR 1
MALMBIJ2 27.05 BOOL  ; ALARM BIJNA OPEN SENSOR 2
MALMDI1 27.06 BOOL  ; ALARM DICHT SENSOR 1
MALMDI2 27.07 BOOL  ; ALARM DICHT SENSOR 2
MALMNOODS H30.00 BOOL  ; ALARM NOODSTOP
MALMOP1 27.02 BOOL  ; ALARM OPEN SENSOR 1
MALMOP2 27.03 BOOL  ; ALARM OPEN SENSOR 2
MALMPAL1 27.00 BOOL  ; PAL ALARM 1
MALMPAL2 27.01 BOOL  ; PAL ALARM 2
MALMW0 170.00 BOOL  ; ALARM IN WOORD HR 30
MALMW1 170.01 BOOL  ; ALARM IN WOORD HR 31
MALMW2 170.02 BOOL  ; ALARM IN WOORD HR 32
MALMW3 170.03 BOOL  ; ALARM IN WOORD HR 33
MALMW4 170.04 BOOL  ; ALARM IN WOORD HR 34
MALMW5 170.05 BOOL  ; ALARM IN WOORD HR 35
MALMW6 170.06 BOOL  ; ALARM IN WOORD HR 36
MALMW7 170.07 BOOL  ; ALARM IN WOORD HR 37
MALMW8 170.08 BOOL  ; ALARM IN WOORD HR 38
MALM_BIJ1 23.04 BOOL  ; ALARM BIJNA OPEN SENSOR 1
MALM_BIJ2 23.05 BOOL  ; ALARM BIJNA OPEN SENSOR 2
MALM_DI1 23.06 BOOL  ; ALARM DICHT SENSOR 1
MALM_DI2 23.07 BOOL  ; ALARM DICHT SENSOR 2
MALM_OP1 23.02 BOOL  ; ALARM OPEN SENSOR 1
MALM_OP2 23.03 BOOL  ; ALARM OPEN SENSOR 2
MALM_PAL1 23.00 BOOL  ; ALARM PAL 1
MALM_PAL2 23.01 BOOL  ; ALARM PAL 2
MALTIJD1 CF113 BOOL  ; SYSTEEMBIT ALTIJD 1
MAL_BEWAK 23.08 BOOL  ; ALARM BEWAKING AANGESPROKEN
MAUTOMAAT H30.01 BOOL  ; ALARM INSTALLATIE AUTOMAAT
MBIT0TMR 26.00 BOOL  ; BIT 0 PRESET STAP TIMER
MBIT10TMR 26.10 BOOL  ; BIT 10 PRESET STAP TIMER
MBIT11TMR 26.11 BOOL  ; BIT 11PRESET STAP TIMER
MBIT12TMR 26.12 BOOL  ; BIT 12 PRESET STAP TIMER
MBIT13TMR 26.13 BOOL  ; BIT 13 PRESET STAP TIMER
MBIT14TMR 26.14 BOOL  ; BIT 14 PRESET STAP TIMER
MBIT15TMR 26.15 BOOL  ; BIT 15 PRESET STAP TIMER
MBIT1TMR 26.01 BOOL  ; BIT 1 PRESET STAP TIMER
MBIT2TMR 26.02 BOOL  ; BIT 2 PRESET STAP TIMER
MBIT3TMR 26.03 BOOL  ; BIT 3 PRESET STAP TIMER
MBIT4TMR 26.04 BOOL  ; BIT 4 PRESET STAP TIMER
MBIT5TMR 26.05 BOOL  ; BIT 5 PRESET STAP TIMER
MBIT6TMR 26.06 BOOL  ; BIT 6 PRESET STAP TIMER
MBIT7TMR 26.07 BOOL  ; BIT 7 PRESET STAP TIMER
MBIT8TMR 26.08 BOOL  ; BIT 8 PRESET STAP TIMER
MBIT9TMR 26.09 BOOL  ; BIT 9 PRESET STAP TIMER
MBLINKER CF101 BOOL  ; BLINK MERKER 5 HZ
MDOORTOEG 25.15 BOOL  ; DOORSTAP TOEGESTAAN
MGELIJK CF006 BOOL  ; IS GELIJK AAN
MI_STAP0 21.00 BOOL  ; STAP 0 (SUB)
MI_STAP1 21.01 BOOL  ; STAP 1 (SUB)
MI_STAP10 21.10 BOOL  ; STAP 10 (SUB)
MI_STAP11 21.11 BOOL  ; STAP 11 (SUB)
MI_STAP12 21.12 BOOL  ; STAP 12 (SUB)
MI_STAP13 21.13 BOOL  ; STAP 13 (SUB)
MI_STAP14 21.14 BOOL  ; STAP 14 (SUB)
MI_STAP15 21.15 BOOL  ; STAP 15 (SUB)
MI_STAP2 21.02 BOOL  ; STAP 2 (SUB)
MI_STAP3 21.03 BOOL  ; STAP 3 (SUB)
MI_STAP4 21.04 BOOL  ; STAP 4 (SUB)
MI_STAP5 21.05 BOOL  ; STAP 5 (SUB)
MI_STAP6 21.06 BOOL  ; STAP 6 (SUB)
MI_STAP7 21.07 BOOL  ; STAP 7 (SUB)
MI_STAP8 21.08 BOOL  ; STAP 8 (SUB)
MI_STAP9 21.09 BOOL  ; STAP 9 (SUB)
MMOTOR_O 24.00 BOOL  ; MOTOR OPENEN (SUB)
MMOTOR_S 24.01 BOOL  ; MOTOR SLUITEN (SUB)
MOSYSTOKE 24.12 BOOL  ; SYSTEEM OKE
MO_STAP0 25.00 BOOL  ; OUTPUT STAP  0 (SUB)
MO_STAP1 25.01 BOOL  ; OUTPUT STAP 1 (SUB)
MO_STAP10 25.10 BOOL  ; OUTPUT STAP 10 (SUB)
MO_STAP11 25.11 BOOL  ; OUTPUT STAP 11 (SUB)
MO_STAP12 25.12 BOOL  ; OUTPUT STAP 12 (SUB)
MO_STAP13 25.13 BOOL  ; OUTPUT STAP 13 (SUB)
MO_STAP14 25.14 BOOL  ; OUTPUT STAP 14 (SUB)
MO_STAP2 25.02 BOOL  ; OUTPUT STAP 2 (SUB)
MO_STAP3 25.03 BOOL  ; OUTPUT STAP 3 (SUB)
MO_STAP4 25.04 BOOL  ; OUTPUT STAP 4 (SUB)
MO_STAP5 25.05 BOOL  ; OUTPUT STAP 5 (SUB)
MO_STAP6 25.06 BOOL  ; OUTPUT STAP 6 (SUB)
MO_STAP7 25.07 BOOL  ; OUTPUT STAP 7  (SUB)
MO_STAP8 25.08 BOOL  ; OUTPUT STAP 8  (SUB)
MO_STAP9 25.09 BOOL  ; OUTPUT STAP 9 (SUB)
MPRTDICHT 24.04 BOOL  ; POORT  IS DICHT
MPRTOPEN 24.03 BOOL  ; POORT  IS OPEN
M_OPENT 24.05 BOOL  ; POORT  IS AAN HET OPENEN
M_PAL 24.02 BOOL  ; PAL OMHOOG STUREN (SUB)
M_SLUIT 24.06 BOOL  ; POORT IS AAN HET SLUITEN
O1L_GREND 101.00 BOOL  ; POORT 1 LINKS VERGRENDELEN
O1L_OPEN 100.00 BOOL  ; POORT 1 LINKS OPENEN
O1L_SLUIT 100.01 BOOL  ; POORT 1 LINKS SLUITEN
O1R_GREND 101.01 BOOL  ; POORT 1 RECHTS VERGRENDELEN
O1R_OPEN 100.02 BOOL  ; POORT 1 RECHTS OPENEN
O1R_SLUIT 100.03 BOOL  ; POORT 1 RECHTS SLUITEN
O2L_GREND 101.02 BOOL  ; POORT 2 LINKS  VERGRENDELEN
O2L_OPEN 100.04 BOOL  ; POORT 2 LINKS OPENEN
O2L_SLUIT 100.05 BOOL  ; POORT 2 LINKS SLUITEN
O2R_GREND 101.03 BOOL  ; POORT 2 RECHTS VERGRENDELEN
O2R_OPEN 100.06 BOOL  ; POORT 2 RECHTS OPENEN
O2R_SLUIT 100.07 BOOL  ; POORT 2 RECHTS SLUITEN
O3L_GREND 101.04 BOOL  ; POORT 3 LINKS VERGRENDELEN
O3L_OPEN 100.08 BOOL  ; POORT 3 LINKS OPENEN
O3L_SLUIT 100.09 BOOL  ; POORT 3 LINKS SLUITEN
O3R_GREND 101.05 BOOL  ; POORT 3 RECHTS VERGRENDELEN
O3R_OPEN 100.10 BOOL  ; POORT 3 RECHTS OPENEN
O3R_SLUIT 100.11 BOOL  ; POORT 3 RECHTS SLUITEN
O4L_GREND 101.06 BOOL  ; POORT 4 LINKS VERGRENDELEN
O4L_OPEN 100.12 BOOL  ; POORT 4 LINKS OPENEN
O4L_SLUIT 100.13 BOOL  ; POORT 4 LINKS SLUITEN
O4R_GREND 101.07 BOOL  ; POORT 4 RECHTS VERGRENDELEN
O4R_OPEN 100.14 BOOL  ; POORT 4 RECHTS OPENEN
O4R_SLUIT 100.15 BOOL  ; POORT 4 RECHTS SLUITEN
O514 101.14 BOOL  ; RESERVE UITGANG 514
O515 101.15 BOOL  ; RESERVE UITGANG 515
OH_IDICHT 101.11 BOOL  ; LAMP POORTJES INGANG DICHT
OH_IOPEN 101.10 BOOL  ; LAMP POORTJES INGANG GEOPEND
OH_READY 101.09 BOOL  ; LAMP READY SIGNAAL
OH_UDICHT 101.13 BOOL  ; LAMP POORTJES UITGANG DICHT
OH_UOPEN 101.12 BOOL  ; LAMP POORTJES UITGANG GEOPEND
OREADY 101.08 BOOL  ; READY SIGNAAL
RALM0OUD D460 CHANNEL  ; REG. ALARM HR 30 VORIGE SCAN
RALM1OUD D461 CHANNEL  ; REG. ALARM HR 31 VORIGE SCAN
RALM2OUD D462 CHANNEL  ; REG. ALARM HR32 VORIGE SCAN
RALM3OUD D463 CHANNEL  ; REG. ALARM HR 33 VORIGE SCAN
RALM4OUD D464 CHANNEL  ; REG. ALARM HR 34 VORIGE SCAN
RALM5OUD D465 CHANNEL  ; REG. ALARM HR 35 VORIGE SCAN
RALM6OUD D466 CHANNEL  ; REG. ALARM HR 36 VORIGE SCAN
RALM7OUD D467 CHANNEL  ; REG. ALARM HR 37 VORIGE SCAN
RALM8OUD D468 CHANNEL  ; REG. ALARM HR 38 VORIGE SCAN
RALMTEMP D459 CHANNEL  ; HULP REG. ALARM
RDALNMR D453 CHANNEL  ; REG. DISPLAY ALARMNUMMER BCD
RDSCHUIF D450 CHANNEL  ; REG. DISPLAY SCHUIFREGISTER
RDTELLER D451 CHANNEL  ; REG. DISPLAY 1 T/M 16
RRALMAKT D452 CHANNEL  ; REG. CONTROLE OF ER IN 1 WOORD EEN ALARM HOOG IS
S9602 96.02 BOOL  ; RESERVE
S9603 96.03 BOOL  ; RESERVE
SOPENEN 20.00 BOOL  ; OPENEN IN/UITGANG (SUB)
SRESET 20.04 BOOL  ; DK RESET BEDIEND (SUB)
SSLUITEN 20.01 BOOL  ; SLUITEN IN/UITGANG (SUB)
SSYSTOKE 20.13 BOOL  ; SYSTEEM OKE (SUB)
START_PULSE 230.01 BOOL  ; START PULSE FROM PUSH BUTTON
S_ALTIJD1 20.14 BOOL  ; ALTIJD 1 BIT  (SUB)
S_BEWAK 20.09 BOOL  ; POORT BEWAKING  (SUB)
S_BIJNA 20.06 BOOL  ; POORT BIJNA DICHT (SUB)
S_DICHT 20.05 BOOL  ; POORT DICHT (SUB)
S_GREND 20.08 BOOL  ; POORT VERGRENDELD  (SUB)
S_OPEN 20.07 BOOL  ; POORT OPEN (SUB)
S_TIMER 20.15 BOOL  ; STAPPENTIMER AFGELOPEN (SUB)
TDISPLAY_PV T206 CHANNEL  ; TIMER OVERBRUG DISPLAY WAARDE
TDISPLAY_Status T0206 BOOL  ; TIMER OVERBRUG DISPLAY WAARDE
TDISPSCRO_PV T207 CHANNEL  ; SCROLLEN ALARMS DISPLAY
TDISPSCRO_Status T0207 BOOL  ; SCROLLEN ALARMS DISPLAY
TIMER_24_VDC_RELAY_01 101 NUMBER  ; TIMER 24 VDC RELAY 01 (ALL RELAY ON)
TIMER_24_VDC_RELAY_02 102 NUMBER  ; TIMER 24 VDC RELAY 02 (ONE RELAY OFF)
TMR_PRG1_PV T31 CHANNEL  ; STAPPENTIMER POORT 1 LINKS
TMR_PRG1_Status T0031 BOOL  ; STAPPENTIMER POORT 1 LINKS
TMR_PRG2_PV T32 CHANNEL  ; STAPPENTIMER POORT 1 RECHTS
TMR_PRG2_Status T0032 BOOL  ; STAPPENTIMER POORT 1 RECHTS
TMR_PRG3_PV T33 CHANNEL  ; STAPPENTIMER POORT 2 LINKS
TMR_PRG3_Status T0033 BOOL  ; STAPPENTIMER POORT 2 LINKS
TMR_PRG4_PV T34 CHANNEL  ; STAPPENTIMER POORT 2 RECHTS
TMR_PRG4_Status T0034 BOOL  ; STAPPENTIMER POORT 2 RECHTS
TMR_PRG5_PV T35 CHANNEL  ; STAPPENTIMER POORT 3 LINKS
TMR_PRG5_Status T0035 BOOL  ; STAPPENTIMER POORT 3 LINKS
TMR_PRG6_PV T36 CHANNEL  ; STAPPENTIMER POORT 3 RECHTS
TMR_PRG6_Status T0036 BOOL  ; STAPPENTIMER POORT 3 RECHTS
TMR_PRG7_PV T37 CHANNEL  ; STAPPENTIMER POORT 4 LINKS
TMR_PRG7_Status T0037 BOOL  ; STAPPENTIMER POORT 4 LINKS
TMR_PRG8_PV T38 CHANNEL  ; STAPPENTIMER POORT 4 RECHTS
TMR_PRG8_Status T0038 BOOL  ; STAPPENTIMER POORT 4 RECHTS
com3_afbreek_show 130.03 BOOL  ; com 3 afbreken show
stop_show 3.03 BOOL  ; afbreken running show

## Program POORTEN (cyclic task 0)
Local symbols
Com3_Alarm_in_Plc3 130.01 BOOL  ; Er is minstens 1 alarm in plc 3 eiland poortjes
Com3_Open_Oever_Poortjes 130.00 BOOL
DK_Open_Oever_Poortjes 3.05 BOOL  ; Open Oever Poortjes

### Section algemeen
; rung 0: PAGODE / *************************************************************************** / Projekt: PAGODE, Besturing poorten        Proj.nr. LvH: 760114 / Locatie: Efteling, Kaatsheuvel. / ***************************************************************************

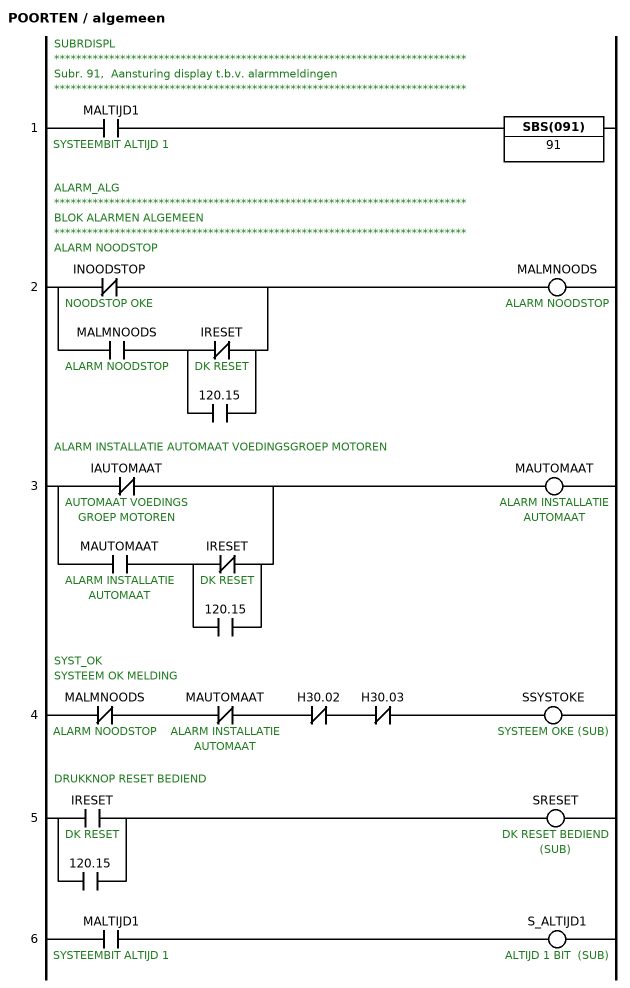
; rung 1: SUBRDISPL / *************************************************************************** / Subr. 91,  Aansturing display t.b.v. alarmmeldingen / ***************************************************************************
LD MALTIJD1  ; SYSTEEMBIT ALTIJD 1
SBS(091) 91
; rung 2: ALARM_ALG / *************************************************************************** / BLOK ALARMEN ALGEMEEN / *************************************************************************** / ALARM NOODSTOP
LDNOT INOODSTOP  ; NOODSTOP OKE
LD MALMNOODS  ; ALARM NOODSTOP
LDNOT IRESET  ; DK RESET
OR 120.15
ANDLD
ORLD
OUT MALMNOODS  ; ALARM NOODSTOP
; rung 3: ALARM INSTALLATIE AUTOMAAT VOEDINGSGROEP MOTOREN
LDNOT IAUTOMAAT  ; AUTOMAAT VOEDINGS GROEP MOTOREN
LD MAUTOMAAT  ; ALARM INSTALLATIE AUTOMAAT
LDNOT IRESET  ; DK RESET
OR 120.15
ANDLD
ORLD
OUT MAUTOMAAT  ; ALARM INSTALLATIE AUTOMAAT
; rung 4: SYST_OK / SYSTEEM OK MELDING
LDNOT MALMNOODS  ; ALARM NOODSTOP
ANDNOT MAUTOMAAT  ; ALARM INSTALLATIE AUTOMAAT
ANDNOT H30.02
ANDNOT H30.03
OUT SSYSTOKE  ; SYSTEEM OKE (SUB)
; rung 5: DRUKKNOP RESET BEDIEND
LD IRESET  ; DK RESET
OR 120.15
OUT SRESET  ; DK RESET BEDIEND (SUB)
; rung 6
LD MALTIJD1  ; SYSTEEMBIT ALTIJD 1
OUT S_ALTIJD1  ; ALTIJD 1 BIT  (SUB)

### Section CONTROL_LINK

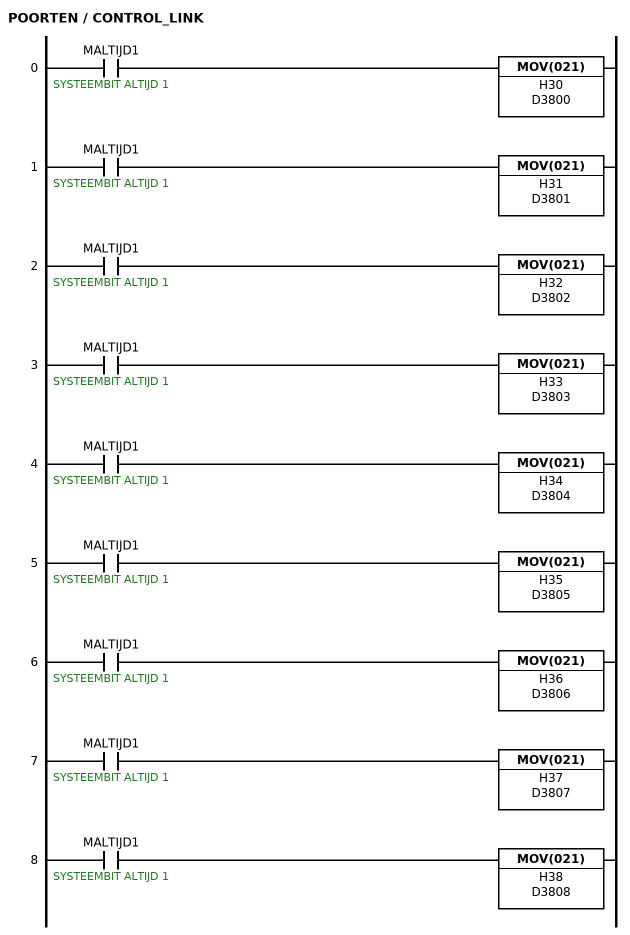
; rung 0
LD MALTIJD1  ; SYSTEEMBIT ALTIJD 1
MOV(021) H30 D3800
; rung 1
LD MALTIJD1  ; SYSTEEMBIT ALTIJD 1
MOV(021) H31 D3801
; rung 2
LD MALTIJD1  ; SYSTEEMBIT ALTIJD 1
MOV(021) H32 D3802
; rung 3
LD MALTIJD1  ; SYSTEEMBIT ALTIJD 1
MOV(021) H33 D3803
; rung 4
LD MALTIJD1  ; SYSTEEMBIT ALTIJD 1
MOV(021) H34 D3804
; rung 5
LD MALTIJD1  ; SYSTEEMBIT ALTIJD 1
MOV(021) H35 D3805
; rung 6
LD MALTIJD1  ; SYSTEEMBIT ALTIJD 1
MOV(021) H36 D3806
; rung 7
LD MALTIJD1  ; SYSTEEMBIT ALTIJD 1
MOV(021) H37 D3807
; rung 8
LD MALTIJD1  ; SYSTEEMBIT ALTIJD 1
MOV(021) H38 D3808

### Section SIGNAAL_DISPLAY

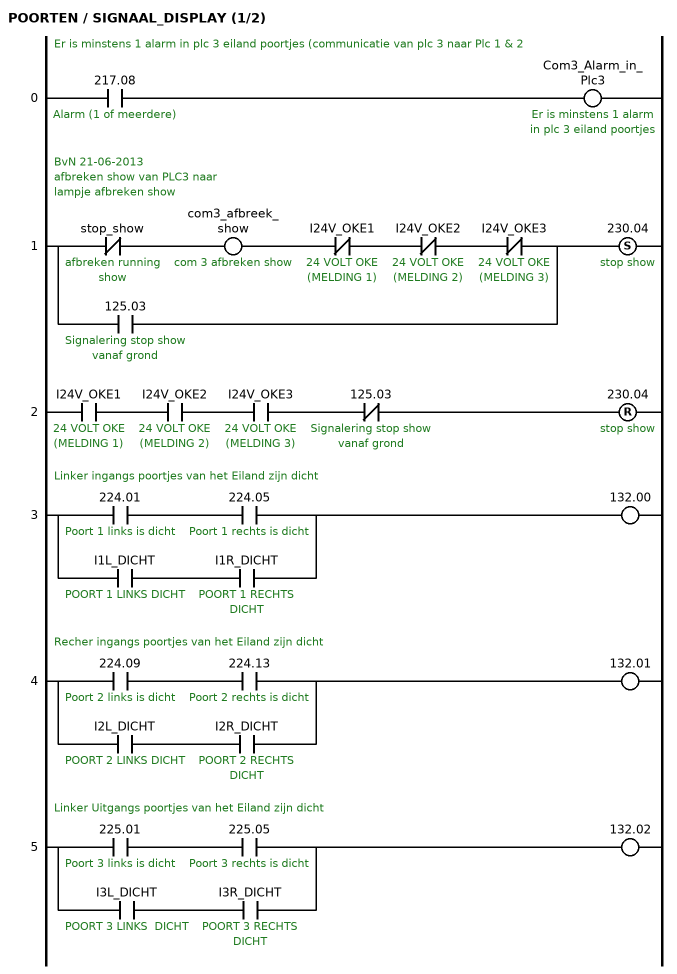
; rung 0: Er is minstens 1 alarm in plc 3 eiland poortjes (communicatie van plc 3 naar Plc 1 & 2
LD 217.08  ; Alarm (1 of meerdere)
OUT Com3_Alarm_in_Plc3  ; Er is minstens 1 alarm in plc 3 eiland poortjes
; rung 1: BvN 21-06-2013 / afbreken show van PLC3 naar / lampje afbreken show
LDNOT stop_show  ; afbreken running show
OUT com3_afbreek_show  ; com 3 afbreken show
ANDNOT I24V_OKE1  ; 24 VOLT OKE (MELDING 1)
ANDNOT I24V_OKE2  ; 24 VOLT OKE (MELDING 2)
ANDNOT I24V_OKE3  ; 24 VOLT OKE (MELDING 3)
OR 125.03  ; Signalering stop show vanaf grond
SET 230.04  ; stop show
; rung 2
LD I24V_OKE1  ; 24 VOLT OKE (MELDING 1)
AND I24V_OKE2  ; 24 VOLT OKE (MELDING 2)
AND I24V_OKE3  ; 24 VOLT OKE (MELDING 3)
ANDNOT 125.03  ; Signalering stop show vanaf grond
RSET 230.04  ; stop show
; rung 3: Linker ingangs poortjes van het Eiland zijn dicht
LD 224.01  ; Poort 1 links is dicht
AND 224.05  ; Poort 1 rechts is dicht
LD I1L_DICHT  ; POORT 1 LINKS DICHT
AND I1R_DICHT  ; POORT 1 RECHTS DICHT
ORLD
OUT 132.00
; rung 4: Recher ingangs poortjes van het Eiland zijn dicht
LD 224.09  ; Poort 2 links is dicht
AND 224.13  ; Poort 2 rechts is dicht
LD I2L_DICHT  ; POORT 2 LINKS DICHT
AND I2R_DICHT  ; POORT 2 RECHTS DICHT
ORLD
OUT 132.01
; rung 5: Linker Uitgangs poortjes van het Eiland zijn dicht
LD 225.01  ; Poort 3 links is dicht
AND 225.05  ; Poort 3 rechts is dicht
LD I3L_DICHT  ; POORT 3 LINKS  DICHT
AND I3R_DICHT  ; POORT 3 RECHTS DICHT
ORLD
OUT 132.02

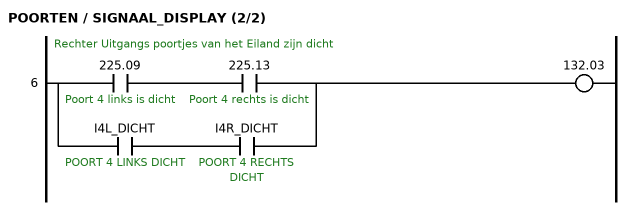
; rung 6: Rechter Uitgangs poortjes van het Eiland zijn dicht
LD 225.09  ; Poort 4 links is dicht
AND 225.13  ; Poort 4 rechts is dicht
LD I4L_DICHT  ; POORT 4 LINKS DICHT
AND I4R_DICHT  ; POORT 4 RECHTS DICHT
ORLD
OUT 132.03

### Section BEDIENING_DISPLAY

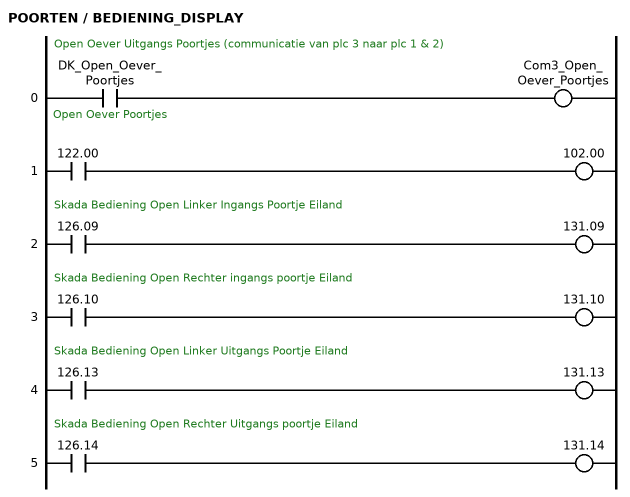
; rung 0: Open Oever Uitgangs Poortjes (communicatie van plc 3 naar plc 1 & 2)
LD DK_Open_Oever_Poortjes  ; Open Oever Poortjes
OUT Com3_Open_Oever_Poortjes
; rung 1
LD 122.00
OUT 102.00
; rung 2: Skada Bediening Open Linker Ingangs Poortje Eiland
LD 126.09
OUT 131.09
; rung 3: Skada Bediening Open Rechter ingangs poortje Eiland
LD 126.10
OUT 131.10
; rung 4: Skada Bediening Open Linker Uitgangs Poortje Eiland
LD 126.13
OUT 131.13
; rung 5: Skada Bediening Open Rechter Uitgangs poortje Eiland
LD 126.14
OUT 131.14

### Section INGANG_POORT_1_L

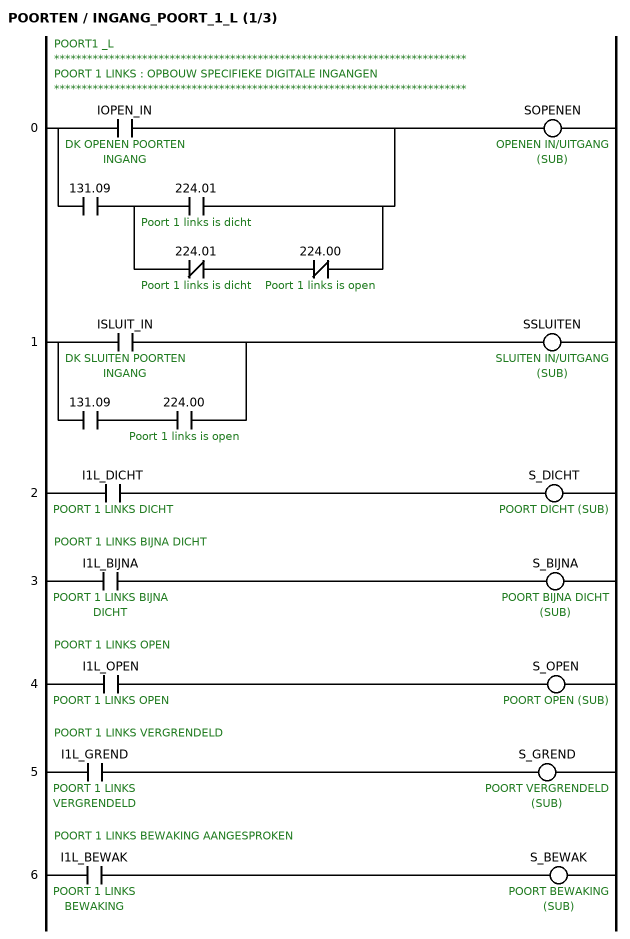
; rung 0: POORT1 _L / *************************************************************************** / POORT 1 LINKS : OPBOUW SPECIFIEKE DIGITALE INGANGEN / ***************************************************************************
LD IOPEN_IN  ; DK OPENEN POORTEN INGANG
LD 131.09
LD 224.01  ; Poort 1 links is dicht
LDNOT 224.01  ; Poort 1 links is dicht
ANDNOT 224.00  ; Poort 1 links is open
ORLD
ANDLD
ORLD
OUT SOPENEN  ; OPENEN IN/UITGANG (SUB)
; rung 1
LD ISLUIT_IN  ; DK SLUITEN POORTEN INGANG
LD 131.09
AND 224.00  ; Poort 1 links is open
ORLD
OUT SSLUITEN  ; SLUITEN IN/UITGANG (SUB)
; rung 2
LD I1L_DICHT  ; POORT 1 LINKS DICHT
OUT S_DICHT  ; POORT DICHT (SUB)
; rung 3: POORT 1 LINKS BIJNA DICHT
LD I1L_BIJNA  ; POORT 1 LINKS BIJNA DICHT
OUT S_BIJNA  ; POORT BIJNA DICHT (SUB)
; rung 4: POORT 1 LINKS OPEN
LD I1L_OPEN  ; POORT 1 LINKS OPEN
OUT S_OPEN  ; POORT OPEN (SUB)
; rung 5: POORT 1 LINKS VERGRENDELD
LD I1L_GREND  ; POORT 1 LINKS VERGRENDELD
OUT S_GREND  ; POORT VERGRENDELD  (SUB)
; rung 6: POORT 1 LINKS BEWAKING AANGESPROKEN
LD I1L_BEWAK  ; POORT 1 LINKS BEWAKING
OUT S_BEWAK  ; POORT BEWAKING  (SUB)

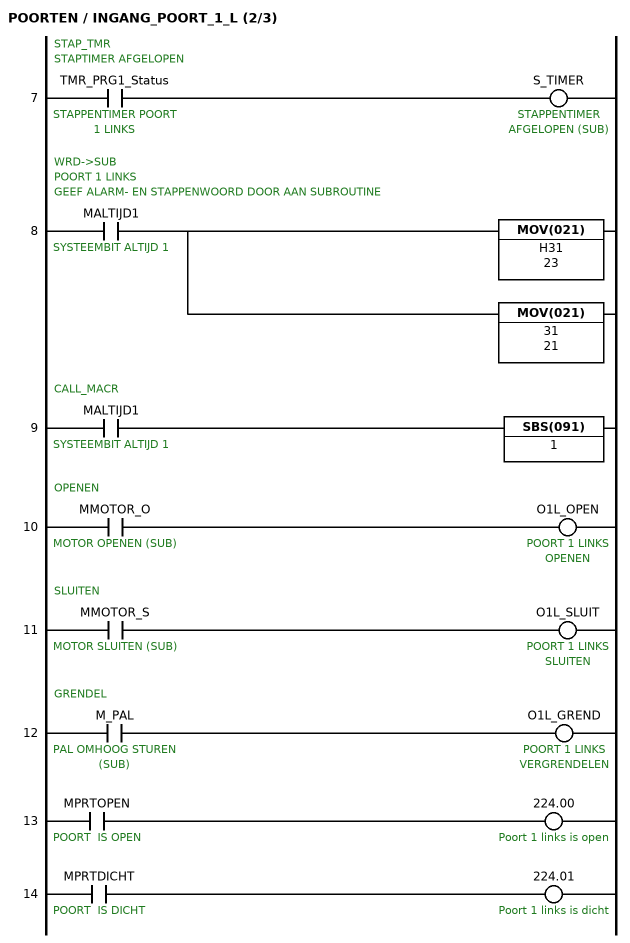
; rung 7: STAP_TMR / STAPTIMER AFGELOPEN
LD TMR_PRG1_Status  ; STAPPENTIMER POORT 1 LINKS
OUT S_TIMER  ; STAPPENTIMER AFGELOPEN (SUB)
; rung 8: WRD->SUB / POORT 1 LINKS / GEEF ALARM- EN STAPPENWOORD DOOR AAN SUBROUTINE
LD MALTIJD1  ; SYSTEEMBIT ALTIJD 1
MOV(021) H31 23
MOV(021) 31 21
; rung 9: CALL_MACR
LD MALTIJD1  ; SYSTEEMBIT ALTIJD 1
SBS(091) 1
; rung 10: OPENEN
LD MMOTOR_O  ; MOTOR OPENEN (SUB)
OUT O1L_OPEN  ; POORT 1 LINKS OPENEN
; rung 11: SLUITEN
LD MMOTOR_S  ; MOTOR SLUITEN (SUB)
OUT O1L_SLUIT  ; POORT 1 LINKS SLUITEN
; rung 12: GRENDEL
LD M_PAL  ; PAL OMHOOG STUREN (SUB)
OUT O1L_GREND  ; POORT 1 LINKS VERGRENDELEN
; rung 13
LD MPRTOPEN  ; POORT  IS OPEN
OUT 224.00  ; Poort 1 links is open
; rung 14
LD MPRTDICHT  ; POORT  IS DICHT
OUT 224.01  ; Poort 1 links is dicht

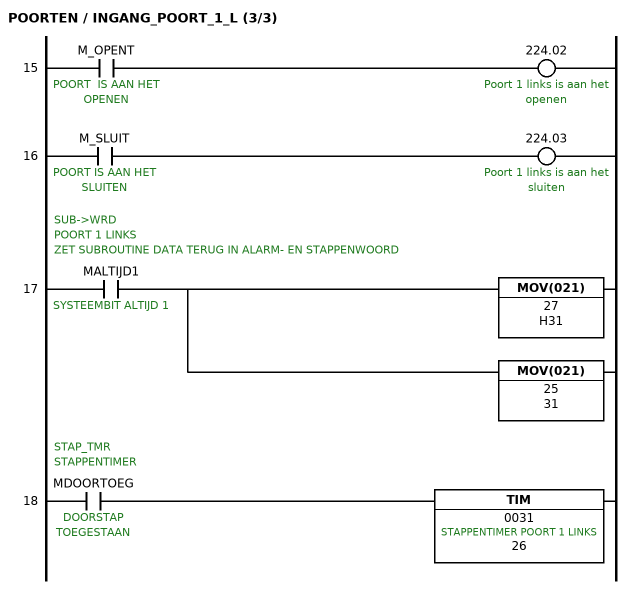
; rung 15
LD M_OPENT  ; POORT  IS AAN HET OPENEN
OUT 224.02  ; Poort 1 links is aan het openen
; rung 16
LD M_SLUIT  ; POORT IS AAN HET SLUITEN
OUT 224.03  ; Poort 1 links is aan het sluiten
; rung 17: SUB->WRD / POORT 1 LINKS / ZET SUBROUTINE DATA TERUG IN ALARM- EN STAPPENWOORD
LD MALTIJD1  ; SYSTEEMBIT ALTIJD 1
MOV(021) 27 H31
MOV(021) 25 31
; rung 18: STAP_TMR / STAPPENTIMER
LD MDOORTOEG  ; DOORSTAP TOEGESTAAN
TIM 0031 26  ; STAPPENTIMER POORT 1 LINKS

### Section INGANG_POORT_1_R

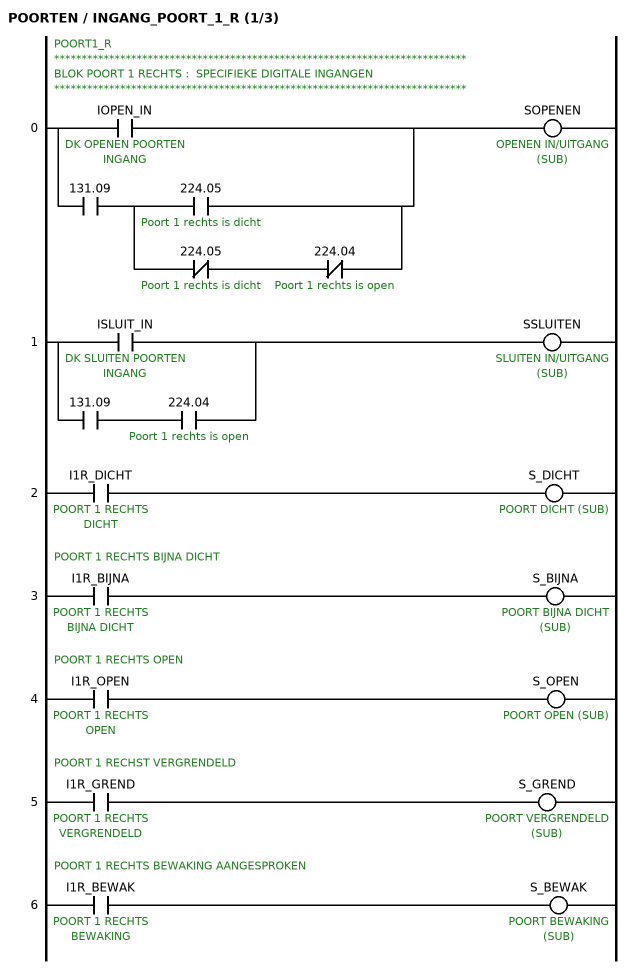
; rung 0: POORT1_R / *************************************************************************** / BLOK POORT 1 RECHTS :  SPECIFIEKE DIGITALE INGANGEN / ***************************************************************************
LD IOPEN_IN  ; DK OPENEN POORTEN INGANG
LD 131.09
LD 224.05  ; Poort 1 rechts is dicht
LDNOT 224.05  ; Poort 1 rechts is dicht
ANDNOT 224.04  ; Poort 1 rechts is open
ORLD
ANDLD
ORLD
OUT SOPENEN  ; OPENEN IN/UITGANG (SUB)
; rung 1
LD ISLUIT_IN  ; DK SLUITEN POORTEN INGANG
LD 131.09
AND 224.04  ; Poort 1 rechts is open
ORLD
OUT SSLUITEN  ; SLUITEN IN/UITGANG (SUB)
; rung 2
LD I1R_DICHT  ; POORT 1 RECHTS DICHT
OUT S_DICHT  ; POORT DICHT (SUB)
; rung 3: POORT 1 RECHTS BIJNA DICHT
LD I1R_BIJNA  ; POORT 1 RECHTS BIJNA DICHT
OUT S_BIJNA  ; POORT BIJNA DICHT (SUB)
; rung 4: POORT 1 RECHTS OPEN
LD I1R_OPEN  ; POORT 1 RECHTS OPEN
OUT S_OPEN  ; POORT OPEN (SUB)
; rung 5: POORT 1 RECHST VERGRENDELD
LD I1R_GREND  ; POORT 1 RECHTS VERGRENDELD
OUT S_GREND  ; POORT VERGRENDELD  (SUB)
; rung 6: POORT 1 RECHTS BEWAKING AANGESPROKEN
LD I1R_BEWAK  ; POORT 1 RECHTS BEWAKING
OUT S_BEWAK  ; POORT BEWAKING  (SUB)

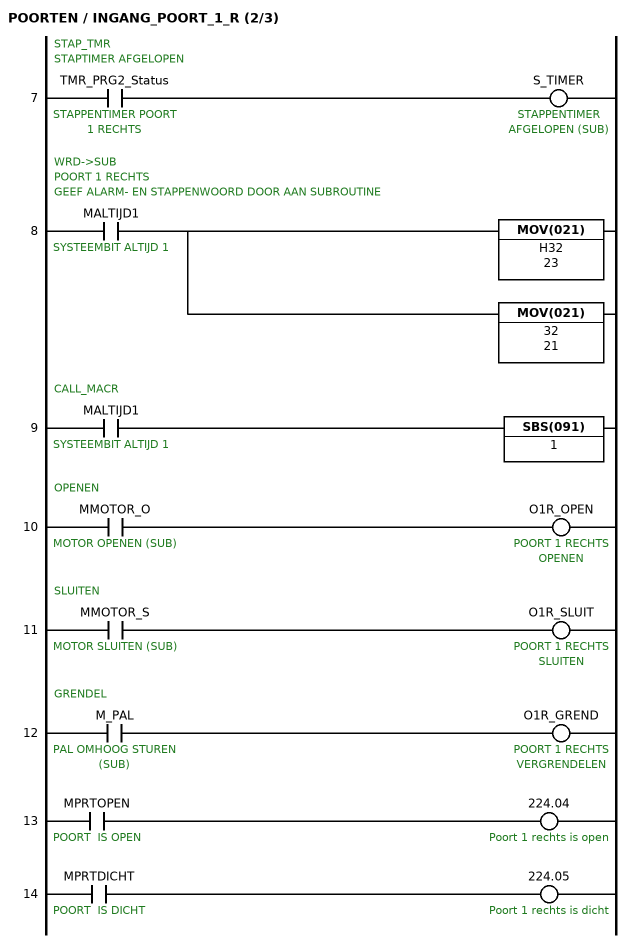
; rung 7: STAP_TMR / STAPTIMER AFGELOPEN
LD TMR_PRG2_Status  ; STAPPENTIMER POORT 1 RECHTS
OUT S_TIMER  ; STAPPENTIMER AFGELOPEN (SUB)
; rung 8: WRD->SUB / POORT 1 RECHTS / GEEF ALARM- EN STAPPENWOORD DOOR AAN SUBROUTINE
LD MALTIJD1  ; SYSTEEMBIT ALTIJD 1
MOV(021) H32 23
MOV(021) 32 21
; rung 9: CALL_MACR
LD MALTIJD1  ; SYSTEEMBIT ALTIJD 1
SBS(091) 1
; rung 10: OPENEN
LD MMOTOR_O  ; MOTOR OPENEN (SUB)
OUT O1R_OPEN  ; POORT 1 RECHTS OPENEN
; rung 11: SLUITEN
LD MMOTOR_S  ; MOTOR SLUITEN (SUB)
OUT O1R_SLUIT  ; POORT 1 RECHTS SLUITEN
; rung 12: GRENDEL
LD M_PAL  ; PAL OMHOOG STUREN (SUB)
OUT O1R_GREND  ; POORT 1 RECHTS VERGRENDELEN
; rung 13
LD MPRTOPEN  ; POORT  IS OPEN
OUT 224.04  ; Poort 1 rechts is open
; rung 14
LD MPRTDICHT  ; POORT  IS DICHT
OUT 224.05  ; Poort 1 rechts is dicht

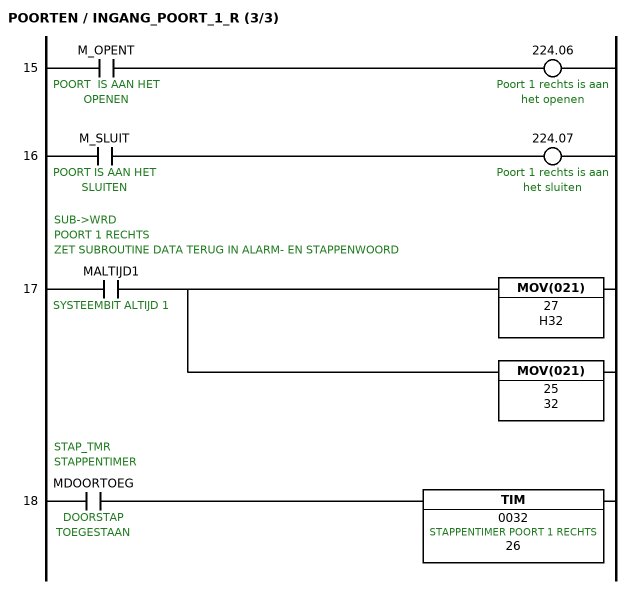
; rung 15
LD M_OPENT  ; POORT  IS AAN HET OPENEN
OUT 224.06  ; Poort 1 rechts is aan het openen
; rung 16
LD M_SLUIT  ; POORT IS AAN HET SLUITEN
OUT 224.07  ; Poort 1 rechts is aan het sluiten
; rung 17: SUB->WRD / POORT 1 RECHTS / ZET SUBROUTINE DATA TERUG IN ALARM- EN STAPPENWOORD
LD MALTIJD1  ; SYSTEEMBIT ALTIJD 1
MOV(021) 27 H32
MOV(021) 25 32
; rung 18: STAP_TMR / STAPPENTIMER
LD MDOORTOEG  ; DOORSTAP TOEGESTAAN
TIM 0032 26  ; STAPPENTIMER POORT 1 RECHTS

### Section INGANG_POORT_2_L

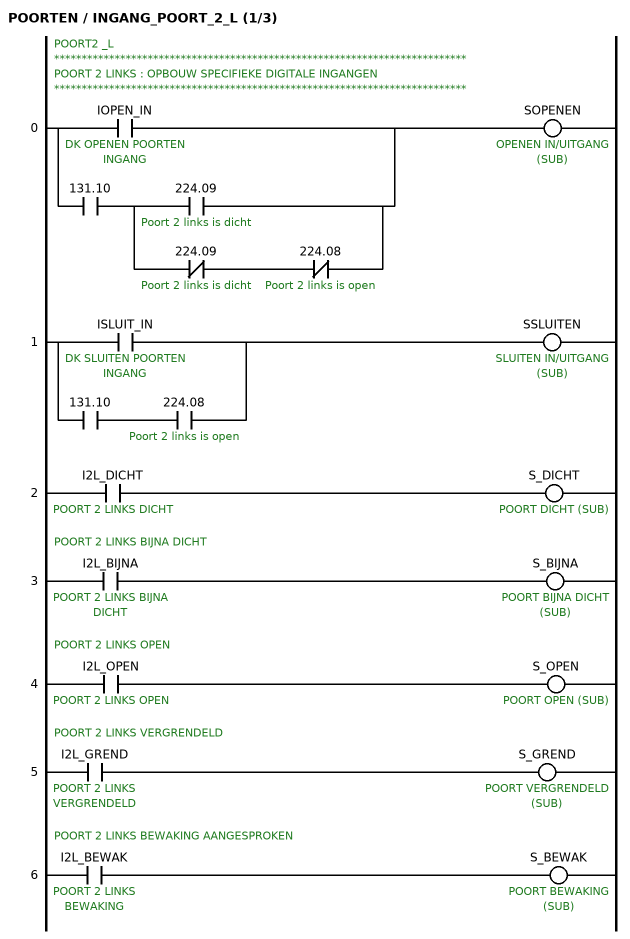
; rung 0: POORT2 _L / *************************************************************************** / POORT 2 LINKS : OPBOUW SPECIFIEKE DIGITALE INGANGEN / ***************************************************************************
LD IOPEN_IN  ; DK OPENEN POORTEN INGANG
LD 131.10
LD 224.09  ; Poort 2 links is dicht
LDNOT 224.09  ; Poort 2 links is dicht
ANDNOT 224.08  ; Poort 2 links is open
ORLD
ANDLD
ORLD
OUT SOPENEN  ; OPENEN IN/UITGANG (SUB)
; rung 1
LD ISLUIT_IN  ; DK SLUITEN POORTEN INGANG
LD 131.10
AND 224.08  ; Poort 2 links is open
ORLD
OUT SSLUITEN  ; SLUITEN IN/UITGANG (SUB)
; rung 2
LD I2L_DICHT  ; POORT 2 LINKS DICHT
OUT S_DICHT  ; POORT DICHT (SUB)
; rung 3: POORT 2 LINKS BIJNA DICHT
LD I2L_BIJNA  ; POORT 2 LINKS BIJNA DICHT
OUT S_BIJNA  ; POORT BIJNA DICHT (SUB)
; rung 4: POORT 2 LINKS OPEN
LD I2L_OPEN  ; POORT 2 LINKS OPEN
OUT S_OPEN  ; POORT OPEN (SUB)
; rung 5: POORT 2 LINKS VERGRENDELD
LD I2L_GREND  ; POORT 2 LINKS VERGRENDELD
OUT S_GREND  ; POORT VERGRENDELD  (SUB)
; rung 6: POORT 2 LINKS BEWAKING AANGESPROKEN
LD I2L_BEWAK  ; POORT 2 LINKS BEWAKING
OUT S_BEWAK  ; POORT BEWAKING  (SUB)

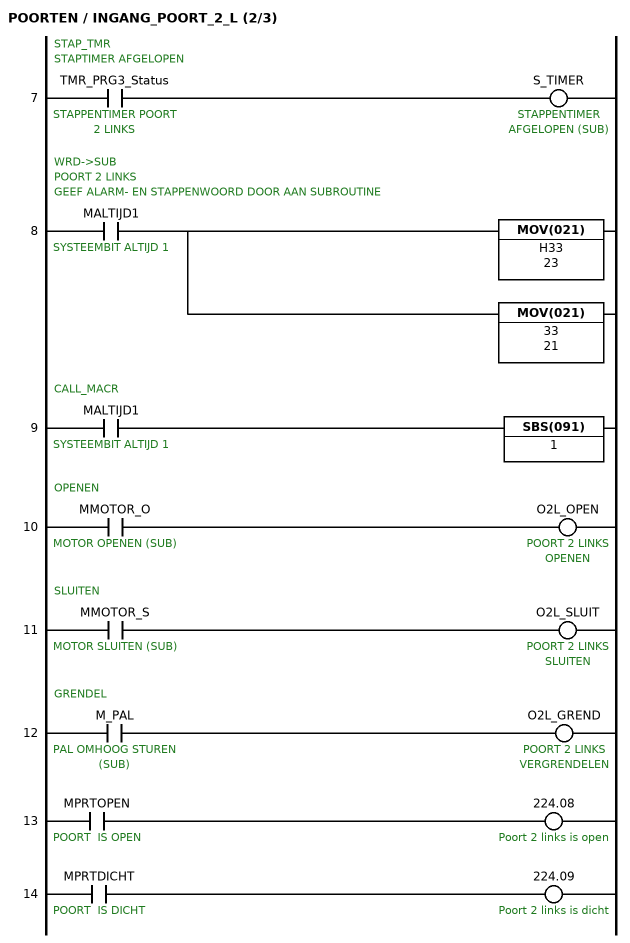
; rung 7: STAP_TMR / STAPTIMER AFGELOPEN
LD TMR_PRG3_Status  ; STAPPENTIMER POORT 2 LINKS
OUT S_TIMER  ; STAPPENTIMER AFGELOPEN (SUB)
; rung 8: WRD->SUB / POORT 2 LINKS / GEEF ALARM- EN STAPPENWOORD DOOR AAN SUBROUTINE
LD MALTIJD1  ; SYSTEEMBIT ALTIJD 1
MOV(021) H33 23
MOV(021) 33 21
; rung 9: CALL_MACR
LD MALTIJD1  ; SYSTEEMBIT ALTIJD 1
SBS(091) 1
; rung 10: OPENEN
LD MMOTOR_O  ; MOTOR OPENEN (SUB)
OUT O2L_OPEN  ; POORT 2 LINKS OPENEN
; rung 11: SLUITEN
LD MMOTOR_S  ; MOTOR SLUITEN (SUB)
OUT O2L_SLUIT  ; POORT 2 LINKS SLUITEN
; rung 12: GRENDEL
LD M_PAL  ; PAL OMHOOG STUREN (SUB)
OUT O2L_GREND  ; POORT 2 LINKS  VERGRENDELEN
; rung 13
LD MPRTOPEN  ; POORT  IS OPEN
OUT 224.08  ; Poort 2 links is open
; rung 14
LD MPRTDICHT  ; POORT  IS DICHT
OUT 224.09  ; Poort 2 links is dicht

